          ;Params IlfProvider=kukaroboter.basistech.inlineforms.movement.spline; Kuka.IsGlobalPoint=False; Kuka.PointName=P254; Kuka.BlendingEnabled=False; Kuka.MoveDataName=CPDAT32; Kuka.VelocityPath=0.1; Kuka.VelocityFieldEnabled=True; Kuka.ColDetectFieldEnabled=True; Kuka.CurrentCDSetIndex=0; Kuka.MovementParameterFieldEnabled=True; IlfCommand=SLIN
          ;ENDFOLD
          SLIN XP254 WITH $VEL = SVEL_CP(0.1, , LCPDAT32), $TOOL = STOOL2(FP254), $BASE = SBASE(FP254.BASE_NO), $IPO_MODE = SIPO_MODE(FP254.IPO_FRAME), $LOAD = SLOAD(FP254.TOOL_NO), $ACC = SACC_CP(LCPDAT32), $ORI_TYPE = SORI_TYP(LCPDAT32), $APO = SAPO(LCPDAT32), $JERK = SJERK(LCPDAT32), $COLLMON_TOL_PRO[1] = USE_CM_PRO_VALUES(0)
          ;ENDFOLD
          ;FOLD Gripper SET [1]Gripper1 State=[2]CERRADA Wait 0.2[s] Check with Strategy 1 ;%{PE}
          ;FOLD Parameters Parameters ;%{h}
          ;Params IlfProvider=GripperTech.GripperSet;setgripper=1;setstate=2;setcont=nocont;waittime=0.2;errorstrategy=1
          ;ENDFOLD
          GRPg_SetStateAndCheck(1, 2, 0.2, 1)
          ;ENDFOLDinitialPosition
          ;FOLD SLIN P154 Vel=0.1 m/s CPDAT33 Tool[1]:SMC Base[0] ;%{PE}
          ;FOLD Parameters ;%{h}s
          ;Params IlfProvider=kukaroboter.basistech.inlineforms.movement.spline; Kuka.IsGlobalPoint=False; Kuka.PointName=P154; Kuka.BlendingEnabled=False; Kuka.MoveDataName=CPDAT33; Kuka.VelocityPath=0.1; Kuka.VelocityFieldEnabled=True; Kuka.ColDetectFieldEnabled=True; Kuka.CurrentCDSetIndex=0; Kuka.MovementParameterFieldEnabled=True; IlfCommand=SLIN
          ;ENDFOLD
          SLIN XP154 WITH $VEL = SVEL_CP(0.1, , LCPDAT33), $TOOL = STOOL2(FP154), $BASE = SBASE(FP154.BASE_NO), $IPO_MODE = SIPO_MODE(FP154.IPO_FRAME), $LOAD = SLOAD(FP154.TOOL_NO), $ACC = SACC_CP(LCPDAT33), $ORI_TYPE = SORI_TYP(LCPDAT33), $APO = SAPO(LCPDAT33), $JERK = SJERK(LCPDAT33), $COLLMON_TOL_PRO[1] = USE_CM_PRO_VALUES(0)
          ;ENDFOLD
          ;FOLD SPTP P500 Vel=100 % PDAT19 Tool[1]:SMC Base[0] ;%{PE}
          ;FOLD Parameters ;%{h}
          ;Params IlfProvider=kukaroboter.basistech.inlineforms.movement.spline; Kuka.IsGlobalPoint=False; Kuka.PointName=P500; Kuka.BlendingEnabled=False; Kuka.MoveDataPtpName=PDAT19; Kuka.VelocityPtp=100; Kuka.VelocityFieldEnabled=True; Kuka.ColDetectFieldEnabled=True; Kuka.CurrentCDSetIndex=0; Kuka.MovementParameterFieldEnabled=True; IlfCommand=SPTP
          ;ENDFOLD
          SPTP XP500 WITH $VEL_AXIS[1] = SVEL_JOINT(100.0), $TOOL = STOOL2(FP500), $BASE = SBASE(FP500.BASE_NO), $IPO_MODE = SIPO_MODE(FP500.IPO_FRAME), $LOAD = SLOAD(FP500.TOOL_NO), $ACC_AXIS[1] = SACC_JOINT(PPDAT19), $APO = SAPO_PTP(PPDAT19), $GEAR_JERK[1] = SGEAR_JERK(PPDAT19), $COLLMON_TOL_PRO[1] = USE_CM_PRO_VALUES(0)
          ;ENDFOLD
          ;FOLD Gripper SET [1]Gripper1 State=[1]ABIERTA Wait 0.2[s] Check with Strategy 1 ;%{PE}
          ;FOLD Parameters Parameters ;%{h}
          ;Params IlfProvider=GripperTech.GripperSet;setgripper=1;setstate=1;setcont=nocont;waittime=0.2;errorstrategy=1
          ;ENDFOLD
          GRPg_SetStateAndCheck(1, 1, 0.2, 1)
          ;ENDFOLD
      ENDIF
      IF eatPosition == 55 THEN
          ;FOLD SPTP P155 Vel=100 % PDAT1 Tool[1]:SMC Base[0] ;%{PE}
          ;FOLD Parameters ;%{h}
          ;Params IlfProvider=kukaroboter.basistech.inlineforms.movement.spline; Kuka.IsGlobalPoint=False; Kuka.PointName=P155; Kuka.BlendingEnabled=False; Kuka.MoveDataPtpName=PDAT1; Kuka.VelocityPtp=100; Kuka.VelocityFieldEnabled=True; Kuka.ColDetectFieldEnabled=True; Kuka.CurrentCDSetIndex=0; Kuka.MovementParameterFieldEnabled=True; IlfCommand=SPTP
          ;ENDFOLD
          SPTP XP155 WITH $VEL_AXIS[1] = SVEL_JOINT(100.0), $TOOL = STOOL2(FP155), $BASE = SBASE(FP155.BASE_NO), $IPO_MODE = SIPO_MODE(FP155.IPO_FRAME), $LOAD = SLOAD(FP155.TOOL_NO), $ACC_AXIS[1] = SACC_JOINT(PPDAT1), $APO = SAPO_PTP(PPDAT1), $GEAR_JERK[1] = SGEAR_JERK(PPDAT1), $COLLMON_TOL_PRO[1] = USE_CM_PRO_VALUES(0)
          ;ENDFOLD
          ;FOLD SLIN P255 Vel=0.1 m/s CPDAT32 Tool[1]:SMC Base[0] ;%{PE}
          ;FOLD Parameters ;%{h}
          ;Params IlfProvider=kukaroboter.basistech.inlineforms.movement.spline; Kuka.IsGlobalPoint=False; Kuka.PointName=P255; Kuka.BlendingEnabled=False; Kuka.MoveDataName=CPDAT32; Kuka.VelocityPath=0.1; Kuka.VelocityFieldEnabled=True; Kuka.ColDetectFieldEnabled=True; Kuka.CurrentCDSetIndex=0; Kuka.MovementParameterFieldEnabled=True; IlfCommand=SLIN
          ;ENDFOLD
          SLIN XP255 WITH $VEL = SVEL_CP(0.1, , LCPDAT32), $TOOL = STOOL2(FP255), $BASE = SBASE(FP255.BASE_NO), $IPO_MODE = SIPO_MODE(FP255.IPO_FRAME), $LOAD = SLOAD(FP255.TOOL_NO), $ACC = SACC_CP(LCPDAT32), $ORI_TYPE = SORI_TYP(LCPDAT32), $APO = SAPO(LCPDAT32), $JERK = SJERK(LCPDAT32), $COLLMON_TOL_PRO[1] = USE_CM_PRO_VALUES(0)
          ;ENDFOLD
          ;FOLD Gripper SET [1]Gripper1 State=[2]CERRADA Wait 0.2[s] Check with Strategy 1 ;%{PE}
          ;FOLD Parameters Parameters ;%{h}
          ;Params IlfProvider=GripperTech.GripperSet;setgripper=1;setstate=2;setcont=nocont;waittime=0.2;errorstrategy=1
          ;ENDFOLD
          GRPg_SetStateAndCheck(1, 2, 0.2, 1)
          ;ENDFOLDinitialPosition
          ;FOLD SLIN P155 Vel=0.1 m/s CPDAT33 Tool[1]:SMC Base[0] ;%{PE}
          ;FOLD Parameters ;%{h}s
          ;Params IlfProvider=kukaroboter.basistech.inlineforms.movement.spline; Kuka.IsGlobalPoint=False; Kuka.PointName=P155; Kuka.BlendingEnabled=False; Kuka.MoveDataName=CPDAT33; Kuka.VelocityPath=0.1; Kuka.VelocityFieldEnabled=True; Kuka.ColDetectFieldEnabled=True; Kuka.CurrentCDSetIndex=0; Kuka.MovementParameterFieldEnabled=True; IlfCommand=SLIN
          ;ENDFOLD
          SLIN XP155 WITH $VEL = SVEL_CP(0.1, , LCPDAT33), $TOOL = STOOL2(FP155), $BASE = SBASE(FP155.BASE_NO), $IPO_MODE = SIPO_MODE(FP155.IPO_FRAME), $LOAD = SLOAD(FP155.TOOL_NO), $ACC = SACC_CP(LCPDAT33), $ORI_TYPE = SORI_TYP(LCPDAT33), $APO = SAPO(LCPDAT33), $JERK = SJERK(LCPDAT33), $COLLMON_TOL_PRO[1] = USE_CM_PRO_VALUES(0)
          ;ENDFOLD
          ;FOLD SPTP P500 Vel=100 % PDAT19 Tool[1]:SMC Base[0] ;%{PE}
          ;FOLD Parameters ;%{h}
          ;Params IlfProvider=kukaroboter.basistech.inlineforms.movement.spline; Kuka.IsGlobalPoint=False; Kuka.PointName=P500; Kuka.BlendingEnabled=False; Kuka.MoveDataPtpName=PDAT19; Kuka.VelocityPtp=100; Kuka.VelocityFieldEnabled=True; Kuka.ColDetectFieldEnabled=True; Kuka.CurrentCDSetIndex=0; Kuka.MovementParameterFieldEnabled=True; IlfCommand=SPTP
          ;ENDFOLD
          SPTP XP500 WITH $VEL_AXIS[1] = SVEL_JOINT(100.0), $TOOL = STOOL2(FP500), $BASE = SBASE(FP500.BASE_NO), $IPO_MODE = SIPO_MODE(FP500.IPO_FRAME), $LOAD = SLOAD(FP500.TOOL_NO), $ACC_AXIS[1] = SACC_JOINT(PPDAT19), $APO = SAPO_PTP(PPDAT19), $GEAR_JERK[1] = SGEAR_JERK(PPDAT19), $COLLMON_TOL_PRO[1] = USE_CM_PRO_VALUES(0)
          ;ENDFOLD
          ;FOLD Gripper SET [1]Gripper1 State=[1]ABIERTA Wait 0.2[s] Check with Strategy 1 ;%{PE}
          ;FOLD Parameters Parameters ;%{h}
          ;Params IlfProvider=GripperTech.GripperSet;setgripper=1;setstate=1;setcont=nocont;waittime=0.2;errorstrategy=1
          ;ENDFOLD
          GRPg_SetStateAndCheck(1, 1, 0.2, 1)
          ;ENDFOLD
      ENDIF
      IF eatPosition == 56 THEN
          ;FOLD SPTP P156 Vel=100 % PDAT1 Tool[1]:SMC Base[0] ;%{PE}
          ;FOLD Parameters ;%{h}
          ;Params IlfProvider=kukaroboter.basistech.inlineforms.movement.spline; Kuka.IsGlobalPoint=False; Kuka.PointName=P156; Kuka.BlendingEnabled=False; Kuka.MoveDataPtpName=PDAT1; Kuka.VelocityPtp=100; Kuka.VelocityFieldEnabled=True; Kuka.ColDetectFieldEnabled=True; Kuka.CurrentCDSetIndex=0; Kuka.MovementParameterFieldEnabled=True; IlfCommand=SPTP
          ;ENDFOLD
          SPTP XP156 WITH $VEL_AXIS[1] = SVEL_JOINT(100.0), $TOOL = STOOL2(FP156), $BASE = SBASE(FP156.BASE_NO), $IPO_MODE = SIPO_MODE(FP156.IPO_FRAME), $LOAD = SLOAD(FP156.TOOL_NO), $ACC_AXIS[1] = SACC_JOINT(PPDAT1), $APO = SAPO_PTP(PPDAT1), $GEAR_JERK[1] = SGEAR_JERK(PPDAT1), $COLLMON_TOL_PRO[1] = USE_CM_PRO_VALUES(0)
          ;ENDFOLD
          ;FOLD SLIN P256 Vel=0.1 m/s CPDAT32 Tool[1]:SMC Base[0] ;%{PE}
          ;FOLD Parameters ;%{h}
          ;Params IlfProvider=kukaroboter.basistech.inlineforms.movement.spline; Kuka.IsGlobalPoint=False; Kuka.PointName=P256; Kuka.BlendingEnabled=False; Kuka.MoveDataName=CPDAT32; Kuka.VelocityPath=0.1; Kuka.VelocityFieldEnabled=True; Kuka.ColDetectFieldEnabled=True; Kuka.CurrentCDSetIndex=0; Kuka.MovementParameterFieldEnabled=True; IlfCommand=SLIN
          ;ENDFOLD
          SLIN XP256 WITH $VEL = SVEL_CP(0.1, , LCPDAT32), $TOOL = STOOL2(FP256), $BASE = SBASE(FP256.BASE_NO), $IPO_MODE = SIPO_MODE(FP256.IPO_FRAME), $LOAD = SLOAD(FP256.TOOL_NO), $ACC = SACC_CP(LCPDAT32), $ORI_TYPE = SORI_TYP(LCPDAT32), $APO = SAPO(LCPDAT32), $JERK = SJERK(LCPDAT32), $COLLMON_TOL_PRO[1] = USE_CM_PRO_VALUES(0)
          ;ENDFOLD
          ;FOLD Gripper SET [1]Gripper1 State=[2]CERRADA Wait 0.2[s] Check with Strategy 1 ;%{PE}
          ;FOLD Parameters Parameters ;%{h}
          ;Params IlfProvider=GripperTech.GripperSet;setgripper=1;setstate=2;setcont=nocont;waittime=0.2;errorstrategy=1
          ;ENDFOLD
          GRPg_SetStateAndCheck(1, 2, 0.2, 1)
          ;ENDFOLDinitialPosition
          ;FOLD SLIN P156 Vel=0.1 m/s CPDAT33 Tool[1]:SMC Base[0] ;%{PE}
          ;FOLD Parameters ;%{h}s
          ;Params IlfProvider=kukaroboter.basistech.inlineforms.movement.spline; Kuka.IsGlobalPoint=False; Kuka.PointName=P156; Kuka.BlendingEnabled=False; Kuka.MoveDataName=CPDAT33; Kuka.VelocityPath=0.1; Kuka.VelocityFieldEnabled=True; Kuka.ColDetectFieldEnabled=True; Kuka.CurrentCDSetIndex=0; Kuka.MovementParameterFieldEnabled=True; IlfCommand=SLIN
          ;ENDFOLD
          SLIN XP156 WITH $VEL = SVEL_CP(0.1, , LCPDAT33), $TOOL = STOOL2(FP156), $BASE = SBASE(FP156.BASE_NO), $IPO_MODE = SIPO_MODE(FP156.IPO_FRAME), $LOAD = SLOAD(FP156.TOOL_NO), $ACC = SACC_CP(LCPDAT33), $ORI_TYPE = SORI_TYP(LCPDAT33), $APO = SAPO(LCPDAT33), $JERK = SJERK(LCPDAT33), $COLLMON_TOL_PRO[1] = USE_CM_PRO_VALUES(0)
          ;ENDFOLD
          ;FOLD SPTP P500 Vel=100 % PDAT19 Tool[1]:SMC Base[0] ;%{PE}
          ;FOLD Parameters ;%{h}
          ;Params IlfProvider=kukaroboter.basistech.inlineforms.movement.spline; Kuka.IsGlobalPoint=False; Kuka.PointName=P500; Kuka.BlendingEnabled=False; Kuka.MoveDataPtpName=PDAT19; Kuka.VelocityPtp=100; Kuka.VelocityFieldEnabled=True; Kuka.ColDetectFieldEnabled=True; Kuka.CurrentCDSetIndex=0; Kuka.MovementParameterFieldEnabled=True; IlfCommand=SPTP
          ;ENDFOLD
          SPTP XP500 WITH $VEL_AXIS[1] = SVEL_JOINT(100.0), $TOOL = STOOL2(FP500), $BASE = SBASE(FP500.BASE_NO), $IPO_MODE = SIPO_MODE(FP500.IPO_FRAME), $LOAD = SLOAD(FP500.TOOL_NO), $ACC_AXIS[1] = SACC_JOINT(PPDAT19), $APO = SAPO_PTP(PPDAT19), $GEAR_JERK[1] = SGEAR_JERK(PPDAT19), $COLLMON_TOL_PRO[1] = USE_CM_PRO_VALUES(0)
          ;ENDFOLD
          ;FOLD Gripper SET [1]Gripper1 State=[1]ABIERTA Wait 0.2[s] Check with Strategy 1 ;%{PE}
          ;FOLD Parameters Parameters ;%{h}
          ;Params IlfProvider=GripperTech.GripperSet;setgripper=1;setstate=1;setcont=nocont;waittime=0.2;errorstrategy=1
          ;ENDFOLD
          GRPg_SetStateAndCheck(1, 1, 0.2, 1)
          ;ENDFOLD
      ENDIF
      IF eatPosition == 57 THEN
          ;FOLD SPTP P157 Vel=100 % PDAT1 Tool[1]:SMC Base[0] ;%{PE}
          ;FOLD Parameters ;%{h}
          ;Params IlfProvider=kukaroboter.basistech.inlineforms.movement.spline; Kuka.IsGlobalPoint=False; Kuka.PointName=P157; Kuka.BlendingEnabled=False; Kuka.MoveDataPtpName=PDAT1; Kuka.VelocityPtp=100; Kuka.VelocityFieldEnabled=True; Kuka.ColDetectFieldEnabled=True; Kuka.CurrentCDSetIndex=0; Kuka.MovementParameterFieldEnabled=True; IlfCommand=SPTP
          ;ENDFOLD
          SPTP XP157 WITH $VEL_AXIS[1] = SVEL_JOINT(100.0), $TOOL = STOOL2(FP157), $BASE = SBASE(FP157.BASE_NO), $IPO_MODE = SIPO_MODE(FP157.IPO_FRAME), $LOAD = SLOAD(FP157.TOOL_NO), $ACC_AXIS[1] = SACC_JOINT(PPDAT1), $APO = SAPO_PTP(PPDAT1), $GEAR_JERK[1] = SGEAR_JERK(PPDAT1), $COLLMON_TOL_PRO[1] = USE_CM_PRO_VALUES(0)
          ;ENDFOLD
          ;FOLD SLIN P257 Vel=0.1 m/s CPDAT32 Tool[1]:SMC Base[0] ;%{PE}
          ;FOLD Parameters ;%{h}
          ;Params IlfProvider=kukaroboter.basistech.inlineforms.movement.spline; Kuka.IsGlobalPoint=False; Kuka.PointName=P257; Kuka.BlendingEnabled=False; Kuka.MoveDataName=CPDAT32; Kuka.VelocityPath=0.1; Kuka.VelocityFieldEnabled=True; Kuka.ColDetectFieldEnabled=True; Kuka.CurrentCDSetIndex=0; Kuka.MovementParameterFieldEnabled=True; IlfCommand=SLIN
          ;ENDFOLD
          SLIN XP257 WITH $VEL = SVEL_CP(0.1, , LCPDAT32), $TOOL = STOOL2(FP257), $BASE = SBASE(FP257.BASE_NO), $IPO_MODE = SIPO_MODE(FP257.IPO_FRAME), $LOAD = SLOAD(FP257.TOOL_NO), $ACC = SACC_CP(LCPDAT32), $ORI_TYPE = SORI_TYP(LCPDAT32), $APO = SAPO(LCPDAT32), $JERK = SJERK(LCPDAT32), $COLLMON_TOL_PRO[1] = USE_CM_PRO_VALUES(0)
          ;ENDFOLD
          ;FOLD Gripper SET [1]Gripper1 State=[2]CERRADA Wait 0.2[s] Check with Strategy 1 ;%{PE}
          ;FOLD Parameters Parameters ;%{h}
          ;Params IlfProvider=GripperTech.GripperSet;setgripper=1;setstate=2;setcont=nocont;waittime=0.2;errorstrategy=1
          ;ENDFOLD
          GRPg_SetStateAndCheck(1, 2, 0.2, 1)
          ;ENDFOLDinitialPosition
          ;FOLD SLIN P157 Vel=0.1 m/s CPDAT33 Tool[1]:SMC Base[0] ;%{PE}
          ;FOLD Parameters ;%{h}s
          ;Params IlfProvider=kukaroboter.basistech.inlineforms.movement.spline; Kuka.IsGlobalPoint=False; Kuka.PointName=P157; Kuka.BlendingEnabled=False; Kuka.MoveDataName=CPDAT33; Kuka.VelocityPath=0.1; Kuka.VelocityFieldEnabled=True; Kuka.ColDetectFieldEnabled=True; Kuka.CurrentCDSetIndex=0; Kuka.MovementParameterFieldEnabled=True; IlfCommand=SLIN
          ;ENDFOLD
          SLIN XP157 WITH $VEL = SVEL_CP(0.1, , LCPDAT33), $TOOL = STOOL2(FP157), $BASE = SBASE(FP157.BASE_NO), $IPO_MODE = SIPO_MODE(FP157.IPO_FRAME), $LOAD = SLOAD(FP157.TOOL_NO), $ACC = SACC_CP(LCPDAT33), $ORI_TYPE = SORI_TYP(LCPDAT33), $APO = SAPO(LCPDAT33), $JERK = SJERK(LCPDAT33), $COLLMON_TOL_PRO[1] = USE_CM_PRO_VALUES(0)
          ;ENDFOLD
          ;FOLD SPTP P500 Vel=100 % PDAT19 Tool[1]:SMC Base[0] ;%{PE}
          ;FOLD Parameters ;%{h}
          ;Params IlfProvider=kukaroboter.basistech.inlineforms.movement.spline; Kuka.IsGlobalPoint=False; Kuka.PointName=P500; Kuka.BlendingEnabled=False; Kuka.MoveDataPtpName=PDAT19; Kuka.VelocityPtp=100; Kuka.VelocityFieldEnabled=True; Kuka.ColDetectFieldEnabled=True; Kuka.CurrentCDSetIndex=0; Kuka.MovementParameterFieldEnabled=True; IlfCommand=SPTP
          ;ENDFOLD
          SPTP XP500 WITH $VEL_AXIS[1] = SVEL_JOINT(100.0), $TOOL = STOOL2(FP500), $BASE = SBASE(FP500.BASE_NO), $IPO_MODE = SIPO_MODE(FP500.IPO_FRAME), $LOAD = SLOAD(FP500.TOOL_NO), $ACC_AXIS[1] = SACC_JOINT(PPDAT19), $APO = SAPO_PTP(PPDAT19), $GEAR_JERK[1] = SGEAR_JERK(PPDAT19), $COLLMON_TOL_PRO[1] = USE_CM_PRO_VALUES(0)
          ;ENDFOLD
          ;FOLD Gripper SET [1]Gripper1 State=[1]ABIERTA Wait 0.2[s] Check with Strategy 1 ;%{PE}
          ;FOLD Parameters Parameters ;%{h}
          ;Params IlfProvider=GripperTech.GripperSet;setgripper=1;setstate=1;setcont=nocont;waittime=0.2;errorstrategy=1
          ;ENDFOLD
          GRPg_SetStateAndCheck(1, 1, 0.2, 1)
          ;ENDFOLD
      ENDIF
      IF eatPosition == 58 THEN
          ;FOLD SPTP P158 Vel=100 % PDAT1 Tool[1]:SMC Base[0] ;%{PE}
          ;FOLD Parameters ;%{h}
          ;Params IlfProvider=kukaroboter.basistech.inlineforms.movement.spline; Kuka.IsGlobalPoint=False; Kuka.PointName=P158; Kuka.BlendingEnabled=False; Kuka.MoveDataPtpName=PDAT1; Kuka.VelocityPtp=100; Kuka.VelocityFieldEnabled=True; Kuka.ColDetectFieldEnabled=True; Kuka.CurrentCDSetIndex=0; Kuka.MovementParameterFieldEnabled=True; IlfCommand=SPTP
          ;ENDFOLD
          SPTP XP158 WITH $VEL_AXIS[1] = SVEL_JOINT(100.0), $TOOL = STOOL2(FP158), $BASE = SBASE(FP158.BASE_NO), $IPO_MODE = SIPO_MODE(FP158.IPO_FRAME), $LOAD = SLOAD(FP158.TOOL_NO), $ACC_AXIS[1] = SACC_JOINT(PPDAT1), $APO = SAPO_PTP(PPDAT1), $GEAR_JERK[1] = SGEAR_JERK(PPDAT1), $COLLMON_TOL_PRO[1] = USE_CM_PRO_VALUES(0)
          ;ENDFOLD
          ;FOLD SLIN P258 Vel=0.1 m/s CPDAT32 Tool[1]:SMC Base[0] ;%{PE}
          ;FOLD Parameters ;%{h}
          ;Params IlfProvider=kukaroboter.basistech.inlineforms.movement.spline; Kuka.IsGlobalPoint=False; Kuka.PointName=P258; Kuka.BlendingEnabled=False; Kuka.MoveDataName=CPDAT32; Kuka.VelocityPath=0.1; Kuka.VelocityFieldEnabled=True; Kuka.ColDetectFieldEnabled=True; Kuka.CurrentCDSetIndex=0; Kuka.MovementParameterFieldEnabled=True; IlfCommand=SLIN
          ;ENDFOLD
          SLIN XP258 WITH $VEL = SVEL_CP(0.1, , LCPDAT32), $TOOL = STOOL2(FP258), $BASE = SBASE(FP258.BASE_NO), $IPO_MODE = SIPO_MODE(FP258.IPO_FRAME), $LOAD = SLOAD(FP258.TOOL_NO), $ACC = SACC_CP(LCPDAT32), $ORI_TYPE = SORI_TYP(LCPDAT32), $APO = SAPO(LCPDAT32), $JERK = SJERK(LCPDAT32), $COLLMON_TOL_PRO[1] = USE_CM_PRO_VALUES(0)
          ;ENDFOLD
          ;FOLD Gripper SET [1]Gripper1 State=[2]CERRADA Wait 0.2[s] Check with Strategy 1 ;%{PE}
          ;FOLD Parameters Parameters ;%{h}
          ;Params IlfProvider=GripperTech.GripperSet;setgripper=1;setstate=2;setcont=nocont;waittime=0.2;errorstrategy=1
          ;ENDFOLD
          GRPg_SetStateAndCheck(1, 2, 0.2, 1)
          ;ENDFOLDinitialPosition
          ;FOLD SLIN P158 Vel=0.1 m/s CPDAT33 Tool[1]:SMC Base[0] ;%{PE}
          ;FOLD Parameters ;%{h}s
          ;Params IlfProvider=kukaroboter.basistech.inlineforms.movement.spline; Kuka.IsGlobalPoint=False; Kuka.PointName=P158; Kuka.BlendingEnabled=False; Kuka.MoveDataName=CPDAT33; Kuka.VelocityPath=0.1; Kuka.VelocityFieldEnabled=True; Kuka.ColDetectFieldEnabled=True; Kuka.CurrentCDSetIndex=0; Kuka.MovementParameterFieldEnabled=True; IlfCommand=SLIN
          ;ENDFOLD
          SLIN XP158 WITH $VEL = SVEL_CP(0.1, , LCPDAT33), $TOOL = STOOL2(FP158), $BASE = SBASE(FP158.BASE_NO), $IPO_MODE = SIPO_MODE(FP158.IPO_FRAME), $LOAD = SLOAD(FP158.TOOL_NO), $ACC = SACC_CP(LCPDAT33), $ORI_TYPE = SORI_TYP(LCPDAT33), $APO = SAPO(LCPDAT33), $JERK = SJERK(LCPDAT33), $COLLMON_TOL_PRO[1] = USE_CM_PRO_VALUES(0)
          ;ENDFOLD
          ;FOLD SPTP P500 Vel=100 % PDAT19 Tool[1]:SMC Base[0] ;%{PE}
          ;FOLD Parameters ;%{h}
          ;Params IlfProvider=kukaroboter.basistech.inlineforms.movement.spline; Kuka.IsGlobalPoint=False; Kuka.PointName=P500; Kuka.BlendingEnabled=False; Kuka.MoveDataPtpName=PDAT19; Kuka.VelocityPtp=100; Kuka.VelocityFieldEnabled=True; Kuka.ColDetectFieldEnabled=True; Kuka.CurrentCDSetIndex=0; Kuka.MovementParameterFieldEnabled=True; IlfCommand=SPTP
          ;ENDFOLD
          SPTP XP500 WITH $VEL_AXIS[1] = SVEL_JOINT(100.0), $TOOL = STOOL2(FP500), $BASE = SBASE(FP500.BASE_NO), $IPO_MODE = SIPO_MODE(FP500.IPO_FRAME), $LOAD = SLOAD(FP500.TOOL_NO), $ACC_AXIS[1] = SACC_JOINT(PPDAT19), $APO = SAPO_PTP(PPDAT19), $GEAR_JERK[1] = SGEAR_JERK(PPDAT19), $COLLMON_TOL_PRO[1] = USE_CM_PRO_VALUES(0)
          ;ENDFOLD
          ;FOLD Gripper SET [1]Gripper1 State=[1]ABIERTA Wait 0.2[s] Check with Strategy 1 ;%{PE}
          ;FOLD Parameters Parameters ;%{h}
          ;Params IlfProvider=GripperTech.GripperSet;setgripper=1;setstate=1;setcont=nocont;waittime=0.2;errorstrategy=1
          ;ENDFOLD
          GRPg_SetStateAndCheck(1, 1, 0.2, 1)
          ;ENDFOLD
      ENDIF
      IF eatPosition == 59 THEN
          ;FOLD SPTP P159 Vel=100 % PDAT1 Tool[1]:SMC Base[0] ;%{PE}
          ;FOLD Parameters ;%{h}
          ;Params IlfProvider=kukaroboter.basistech.inlineforms.movement.spline; Kuka.IsGlobalPoint=False; Kuka.PointName=P159; Kuka.BlendingEnabled=False; Kuka.MoveDataPtpName=PDAT1; Kuka.VelocityPtp=100; Kuka.VelocityFieldEnabled=True; Kuka.ColDetectFieldEnabled=True; Kuka.CurrentCDSetIndex=0; Kuka.MovementParameterFieldEnabled=True; IlfCommand=SPTP
          ;ENDFOLD
          SPTP XP159 WITH $VEL_AXIS[1] = SVEL_JOINT(100.0), $TOOL = STOOL2(FP159), $BASE = SBASE(FP159.BASE_NO), $IPO_MODE = SIPO_MODE(FP159.IPO_FRAME), $LOAD = SLOAD(FP159.TOOL_NO), $ACC_AXIS[1] = SACC_JOINT(PPDAT1), $APO = SAPO_PTP(PPDAT1), $GEAR_JERK[1] = SGEAR_JERK(PPDAT1), $COLLMON_TOL_PRO[1] = USE_CM_PRO_VALUES(0)
          ;ENDFOLD
          ;FOLD SLIN P259 Vel=0.1 m/s CPDAT32 Tool[1]:SMC Base[0] ;%{PE}
          ;FOLD Parameters ;%{h}
          ;Params IlfProvider=kukaroboter.basistech.inlineforms.movement.spline; Kuka.IsGlobalPoint=False; Kuka.PointName=P259; Kuka.BlendingEnabled=False; Kuka.MoveDataName=CPDAT32; Kuka.VelocityPath=0.1; Kuka.VelocityFieldEnabled=True; Kuka.ColDetectFieldEnabled=True; Kuka.CurrentCDSetIndex=0; Kuka.MovementParameterFieldEnabled=True; IlfCommand=SLIN
          ;ENDFOLD
          SLIN XP259 WITH $VEL = SVEL_CP(0.1, , LCPDAT32), $TOOL = STOOL2(FP259), $BASE = SBASE(FP259.BASE_NO), $IPO_MODE = SIPO_MODE(FP259.IPO_FRAME), $LOAD = SLOAD(FP259.TOOL_NO), $ACC = SACC_CP(LCPDAT32), $ORI_TYPE = SORI_TYP(LCPDAT32), $APO = SAPO(LCPDAT32), $JERK = SJERK(LCPDAT32), $COLLMON_TOL_PRO[1] = USE_CM_PRO_VALUES(0)
          ;ENDFOLD
          ;FOLD Gripper SET [1]Gripper1 State=[2]CERRADA Wait 0.2[s] Check with Strategy 1 ;%{PE}
          ;FOLD Parameters Parameters ;%{h}
          ;Params IlfProvider=GripperTech.GripperSet;setgripper=1;setstate=2;setcont=nocont;waittime=0.2;errorstrategy=1
          ;ENDFOLD
          GRPg_SetStateAndCheck(1, 2, 0.2, 1)
          ;ENDFOLDinitialPosition
          ;FOLD SLIN P159 Vel=0.1 m/s CPDAT33 Tool[1]:SMC Base[0] ;%{PE}
          ;FOLD Parameters ;%{h}s
          ;Params IlfProvider=kukaroboter.basistech.inlineforms.movement.spline; Kuka.IsGlobalPoint=False; Kuka.PointName=P159; Kuka.BlendingEnabled=False; Kuka.MoveDataName=CPDAT33; Kuka.VelocityPath=0.1; Kuka.VelocityFieldEnabled=True; Kuka.ColDetectFieldEnabled=True; Kuka.CurrentCDSetIndex=0; Kuka.MovementParameterFieldEnabled=True; IlfCommand=SLIN
          ;ENDFOLD
          SLIN XP159 WITH $VEL = SVEL_CP(0.1, , LCPDAT33), $TOOL = STOOL2(FP159), $BASE = SBASE(FP159.BASE_NO), $IPO_MODE = SIPO_MODE(FP159.IPO_FRAME), $LOAD = SLOAD(FP159.TOOL_NO), $ACC = SACC_CP(LCPDAT33), $ORI_TYPE = SORI_TYP(LCPDAT33), $APO = SAPO(LCPDAT33), $JERK = SJERK(LCPDAT33), $COLLMON_TOL_PRO[1] = USE_CM_PRO_VALUES(0)
          ;ENDFOLD
          ;FOLD SPTP P500 Vel=100 % PDAT19 Tool[1]:SMC Base[0] ;%{PE}
          ;FOLD Parameters ;%{h}
          ;Params IlfProvider=kukaroboter.basistech.inlineforms.movement.spline; Kuka.IsGlobalPoint=False; Kuka.PointName=P500; Kuka.BlendingEnabled=False; Kuka.MoveDataPtpName=PDAT19; Kuka.VelocityPtp=100; Kuka.VelocityFieldEnabled=True; Kuka.ColDetectFieldEnabled=True; Kuka.CurrentCDSetIndex=0; Kuka.MovementParameterFieldEnabled=True; IlfCommand=SPTP
          ;ENDFOLD
          SPTP XP500 WITH $VEL_AXIS[1] = SVEL_JOINT(100.0), $TOOL = STOOL2(FP500), $BASE = SBASE(FP500.BASE_NO), $IPO_MODE = SIPO_MODE(FP500.IPO_FRAME), $LOAD = SLOAD(FP500.TOOL_NO), $ACC_AXIS[1] = SACC_JOINT(PPDAT19), $APO = SAPO_PTP(PPDAT19), $GEAR_JERK[1] = SGEAR_JERK(PPDAT19), $COLLMON_TOL_PRO[1] = USE_CM_PRO_VALUES(0)
          ;ENDFOLD
          ;FOLD Gripper SET [1]Gripper1 State=[1]ABIERTA Wait 0.2[s] Check with Strategy 1 ;%{PE}
          ;FOLD Parameters Parameters ;%{h}
          ;Params IlfProvider=GripperTech.GripperSet;setgripper=1;setstate=1;setcont=nocont;waittime=0.2;errorstrategy=1
          ;ENDFOLD
          GRPg_SetStateAndCheck(1, 1, 0.2, 1)
          ;ENDFOLD
      ENDIF
      IF eatPosition == 60 THEN
          ;FOLD SPTP P160 Vel=100 % PDAT1 Tool[1]:SMC Base[0] ;%{PE}
          ;FOLD Parameters ;%{h}
          ;Params IlfProvider=kukaroboter.basistech.inlineforms.movement.spline; Kuka.IsGlobalPoint=False; Kuka.PointName=P160; Kuka.BlendingEnabled=False; Kuka.MoveDataPtpName=PDAT1; Kuka.VelocityPtp=100; Kuka.VelocityFieldEnabled=True; Kuka.ColDetectFieldEnabled=True; Kuka.CurrentCDSetIndex=0; Kuka.MovementParameterFieldEnabled=True; IlfCommand=SPTP
          ;ENDFOLD
          SPTP XP160 WITH $VEL_AXIS[1] = SVEL_JOINT(100.0), $TOOL = STOOL2(FP160), $BASE = SBASE(FP160.BASE_NO), $IPO_MODE = SIPO_MODE(FP160.IPO_FRAME), $LOAD = SLOAD(FP160.TOOL_NO), $ACC_AXIS[1] = SACC_JOINT(PPDAT1), $APO = SAPO_PTP(PPDAT1), $GEAR_JERK[1] = SGEAR_JERK(PPDAT1), $COLLMON_TOL_PRO[1] = USE_CM_PRO_VALUES(0)
          ;ENDFOLD
          ;FOLD SLIN P260 Vel=0.1 m/s CPDAT32 Tool[1]:SMC Base[0] ;%{PE}
          ;FOLD Parameters ;%{h}
          ;Params IlfProvider=kukaroboter.basistech.inlineforms.movement.spline; Kuka.IsGlobalPoint=False; Kuka.PointName=P260; Kuka.BlendingEnabled=False; Kuka.MoveDataName=CPDAT32; Kuka.VelocityPath=0.1; Kuka.VelocityFieldEnabled=True; Kuka.ColDetectFieldEnabled=True; Kuka.CurrentCDSetIndex=0; Kuka.MovementParameterFieldEnabled=True; IlfCommand=SLIN
          ;ENDFOLD
          SLIN XP260 WITH $VEL = SVEL_CP(0.1, , LCPDAT32), $TOOL = STOOL2(FP260), $BASE = SBASE(FP260.BASE_NO), $IPO_MODE = SIPO_MODE(FP260.IPO_FRAME), $LOAD = SLOAD(FP260.TOOL_NO), $ACC = SACC_CP(LCPDAT32), $ORI_TYPE = SORI_TYP(LCPDAT32), $APO = SAPO(LCPDAT32), $JERK = SJERK(LCPDAT32), $COLLMON_TOL_PRO[1] = USE_CM_PRO_VALUES(0)
          ;ENDFOLD
          ;FOLD Gripper SET [1]Gripper1 State=[2]CERRADA Wait 0.2[s] Check with Strategy 1 ;%{PE}
          ;FOLD Parameters Parameters ;%{h}
          ;Params IlfProvider=GripperTech.GripperSet;setgripper=1;setstate=2;setcont=nocont;waittime=0.2;errorstrategy=1
          ;ENDFOLD
          GRPg_SetStateAndCheck(1, 2, 0.2, 1)
          ;ENDFOLDinitialPosition
          ;FOLD SLIN P160 Vel=0.1 m/s CPDAT33 Tool[1]:SMC Base[0] ;%{PE}
          ;FOLD Parameters ;%{h}s
          ;Params IlfProvider=kukaroboter.basistech.inlineforms.movement.spline; Kuka.IsGlobalPoint=False; Kuka.PointName=P160; Kuka.BlendingEnabled=False; Kuka.MoveDataName=CPDAT33; Kuka.VelocityPath=0.1; Kuka.VelocityFieldEnabled=True; Kuka.ColDetectFieldEnabled=True; Kuka.CurrentCDSetIndex=0; Kuka.MovementParameterFieldEnabled=True; IlfCommand=SLIN
          ;ENDFOLD
          SLIN XP160 WITH $VEL = SVEL_CP(0.1, , LCPDAT33), $TOOL = STOOL2(FP160), $BASE = SBASE(FP160.BASE_NO), $IPO_MODE = SIPO_MODE(FP160.IPO_FRAME), $LOAD = SLOAD(FP160.TOOL_NO), $ACC = SACC_CP(LCPDAT33), $ORI_TYPE = SORI_TYP(LCPDAT33), $APO = SAPO(LCPDAT33), $JERK = SJERK(LCPDAT33), $COLLMON_TOL_PRO[1] = USE_CM_PRO_VALUES(0)
          ;ENDFOLD
          ;FOLD SPTP P500 Vel=100 % PDAT19 Tool[1]:SMC Base[0] ;%{PE}
          ;FOLD Parameters ;%{h}
          ;Params IlfProvider=kukaroboter.basistech.inlineforms.movement.spline; Kuka.IsGlobalPoint=False; Kuka.PointName=P500; Kuka.BlendingEnabled=False; Kuka.MoveDataPtpName=PDAT19; Kuka.VelocityPtp=100; Kuka.VelocityFieldEnabled=True; Kuka.ColDetectFieldEnabled=True; Kuka.CurrentCDSetIndex=0; Kuka.MovementParameterFieldEnabled=True; IlfCommand=SPTP
          ;ENDFOLD
          SPTP XP500 WITH $VEL_AXIS[1] = SVEL_JOINT(100.0), $TOOL = STOOL2(FP500), $BASE = SBASE(FP500.BASE_NO), $IPO_MODE = SIPO_MODE(FP500.IPO_FRAME), $LOAD = SLOAD(FP500.TOOL_NO), $ACC_AXIS[1] = SACC_JOINT(PPDAT19), $APO = SAPO_PTP(PPDAT19), $GEAR_JERK[1] = SGEAR_JERK(PPDAT19), $COLLMON_TOL_PRO[1] = USE_CM_PRO_VALUES(0)
          ;ENDFOLD
          ;FOLD Gripper SET [1]Gripper1 State=[1]ABIERTA Wait 0.2[s] Check with Strategy 1 ;%{PE}
          ;FOLD Parameters Parameters ;%{h}
          ;Params IlfProvider=GripperTech.GripperSet;setgripper=1;setstate=1;setcont=nocont;waittime=0.2;errorstrategy=1
          ;ENDFOLD
          GRPg_SetStateAndCheck(1, 1, 0.2, 1)
          ;ENDFOLD
      ENDIF
      IF eatPosition == 61 THEN
          ;FOLD SPTP P161 Vel=100 % PDAT1 Tool[1]:SMC Base[0] ;%{PE}
          ;FOLD Parameters ;%{h}
          ;Params IlfProvider=kukaroboter.basistech.inlineforms.movement.spline; Kuka.IsGlobalPoint=False; Kuka.PointName=P161; Kuka.BlendingEnabled=False; Kuka.MoveDataPtpName=PDAT1; Kuka.VelocityPtp=100; Kuka.VelocityFieldEnabled=True; Kuka.ColDetectFieldEnabled=True; Kuka.CurrentCDSetIndex=0; Kuka.MovementParameterFieldEnabled=True; IlfCommand=SPTP
          ;ENDFOLD
          SPTP XP161 WITH $VEL_AXIS[1] = SVEL_JOINT(100.0), $TOOL = STOOL2(FP161), $BASE = SBASE(FP161.BASE_NO), $IPO_MODE = SIPO_MODE(FP161.IPO_FRAME), $LOAD = SLOAD(FP161.TOOL_NO), $ACC_AXIS[1] = SACC_JOINT(PPDAT1), $APO = SAPO_PTP(PPDAT1), $GEAR_JERK[1] = SGEAR_JERK(PPDAT1), $COLLMON_TOL_PRO[1] = USE_CM_PRO_VALUES(0)
          ;ENDFOLD
          ;FOLD SLIN P261 Vel=0.1 m/s CPDAT32 Tool[1]:SMC Base[0] ;%{PE}
          ;FOLD Parameters ;%{h}
          ;Params IlfProvider=kukaroboter.basistech.inlineforms.movement.spline; Kuka.IsGlobalPoint=False; Kuka.PointName=P261; Kuka.BlendingEnabled=False; Kuka.MoveDataName=CPDAT32; Kuka.VelocityPath=0.1; Kuka.VelocityFieldEnabled=True; Kuka.ColDetectFieldEnabled=True; Kuka.CurrentCDSetIndex=0; Kuka.MovementParameterFieldEnabled=True; IlfCommand=SLIN
          ;ENDFOLD
          SLIN XP261 WITH $VEL = SVEL_CP(0.1, , LCPDAT32), $TOOL = STOOL2(FP261), $BASE = SBASE(FP261.BASE_NO), $IPO_MODE = SIPO_MODE(FP261.IPO_FRAME), $LOAD = SLOAD(FP261.TOOL_NO), $ACC = SACC_CP(LCPDAT32), $ORI_TYPE = SORI_TYP(LCPDAT32), $APO = SAPO(LCPDAT32), $JERK = SJERK(LCPDAT32), $COLLMON_TOL_PRO[1] = USE_CM_PRO_VALUES(0)
          ;ENDFOLD
          ;FOLD Gripper SET [1]Gripper1 State=[2]CERRADA Wait 0.2[s] Check with Strategy 1 ;%{PE}
          ;FOLD Parameters Parameters ;%{h}
          ;Params IlfProvider=GripperTech.GripperSet;setgripper=1;setstate=2;setcont=nocont;waittime=0.2;errorstrategy=1
          ;ENDFOLD
          GRPg_SetStateAndCheck(1, 2, 0.2, 1)
          ;ENDFOLDinitialPosition
          ;FOLD SLIN P161 Vel=0.1 m/s CPDAT33 Tool[1]:SMC Base[0] ;%{PE}
          ;FOLD Parameters ;%{h}s
          ;Params IlfProvider=kukaroboter.basistech.inlineforms.movement.spline; Kuka.IsGlobalPoint=False; Kuka.PointName=P161; Kuka.BlendingEnabled=False; Kuka.MoveDataName=CPDAT33; Kuka.VelocityPath=0.1; Kuka.VelocityFieldEnabled=True; Kuka.ColDetectFieldEnabled=True; Kuka.CurrentCDSetIndex=0; Kuka.MovementParameterFieldEnabled=True; IlfCommand=SLIN
          ;ENDFOLD
          SLIN XP161 WITH $VEL = SVEL_CP(0.1, , LCPDAT33), $TOOL = STOOL2(FP161), $BASE = SBASE(FP161.BASE_NO), $IPO_MODE = SIPO_MODE(FP161.IPO_FRAME), $LOAD = SLOAD(FP161.TOOL_NO), $ACC = SACC_CP(LCPDAT33), $ORI_TYPE = SORI_TYP(LCPDAT33), $APO = SAPO(LCPDAT33), $JERK = SJERK(LCPDAT33), $COLLMON_TOL_PRO[1] = USE_CM_PRO_VALUES(0)
          ;ENDFOLD
          ;FOLD SPTP P500 Vel=100 % PDAT19 Tool[1]:SMC Base[0] ;%{PE}
          ;FOLD Parameters ;%{h}
          ;Params IlfProvider=kukaroboter.basistech.inlineforms.movement.spline; Kuka.IsGlobalPoint=False; Kuka.PointName=P500; Kuka.BlendingEnabled=False; Kuka.MoveDataPtpName=PDAT19; Kuka.VelocityPtp=100; Kuka.VelocityFieldEnabled=True; Kuka.ColDetectFieldEnabled=True; Kuka.CurrentCDSetIndex=0; Kuka.MovementParameterFieldEnabled=True; IlfCommand=SPTP
          ;ENDFOLD
          SPTP XP500 WITH $VEL_AXIS[1] = SVEL_JOINT(100.0), $TOOL = STOOL2(FP500), $BASE = SBASE(FP500.BASE_NO), $IPO_MODE = SIPO_MODE(FP500.IPO_FRAME), $LOAD = SLOAD(FP500.TOOL_NO), $ACC_AXIS[1] = SACC_JOINT(PPDAT19), $APO = SAPO_PTP(PPDAT19), $GEAR_JERK[1] = SGEAR_JERK(PPDAT19), $COLLMON_TOL_PRO[1] = USE_CM_PRO_VALUES(0)
          ;ENDFOLD
          ;FOLD Gripper SET [1]Gripper1 State=[1]ABIERTA Wait 0.2[s] Check with Strategy 1 ;%{PE}
          ;FOLD Parameters Parameters ;%{h}
          ;Params IlfProvider=GripperTech.GripperSet;setgripper=1;setstate=1;setcont=nocont;waittime=0.2;errorstrategy=1
          ;ENDFOLD
          GRPg_SetStateAndCheck(1, 1, 0.2, 1)
          ;ENDFOLD
      ENDIF
      IF eatPosition == 62 THEN
          ;FOLD SPTP P162 Vel=100 % PDAT1 Tool[1]:SMC Base[0] ;%{PE}
          ;FOLD Parameters ;%{h}
          ;Params IlfProvider=kukaroboter.basistech.inlineforms.movement.spline; Kuka.IsGlobalPoint=False; Kuka.PointName=P162; Kuka.BlendingEnabled=False; Kuka.MoveDataPtpName=PDAT1; Kuka.VelocityPtp=100; Kuka.VelocityFieldEnabled=True; Kuka.ColDetectFieldEnabled=True; Kuka.CurrentCDSetIndex=0; Kuka.MovementParameterFieldEnabled=True; IlfCommand=SPTP
          ;ENDFOLD
          SPTP XP162 WITH $VEL_AXIS[1] = SVEL_JOINT(100.0), $TOOL = STOOL2(FP162), $BASE = SBASE(FP162.BASE_NO), $IPO_MODE = SIPO_MODE(FP162.IPO_FRAME), $LOAD = SLOAD(FP162.TOOL_NO), $ACC_AXIS[1] = SACC_JOINT(PPDAT1), $APO = SAPO_PTP(PPDAT1), $GEAR_JERK[1] = SGEAR_JERK(PPDAT1), $COLLMON_TOL_PRO[1] = USE_CM_PRO_VALUES(0)
          ;ENDFOLD
          ;FOLD SLIN P262 Vel=0.1 m/s CPDAT32 Tool[1]:SMC Base[0] ;%{PE}
          ;FOLD Parameters ;%{h}
          ;Params IlfProvider=kukaroboter.basistech.inlineforms.movement.spline; Kuka.IsGlobalPoint=False; Kuka.PointName=P262; Kuka.BlendingEnabled=False; Kuka.MoveDataName=CPDAT32; Kuka.VelocityPath=0.1; Kuka.VelocityFieldEnabled=True; Kuka.ColDetectFieldEnabled=True; Kuka.CurrentCDSetIndex=0; Kuka.MovementParameterFieldEnabled=True; IlfCommand=SLIN
          ;ENDFOLD
          SLIN XP262 WITH $VEL = SVEL_CP(0.1, , LCPDAT32), $TOOL = STOOL2(FP262), $BASE = SBASE(FP262.BASE_NO), $IPO_MODE = SIPO_MODE(FP262.IPO_FRAME), $LOAD = SLOAD(FP262.TOOL_NO), $ACC = SACC_CP(LCPDAT32), $ORI_TYPE = SORI_TYP(LCPDAT32), $APO = SAPO(LCPDAT32), $JERK = SJERK(LCPDAT32), $COLLMON_TOL_PRO[1] = USE_CM_PRO_VALUES(0)
          ;ENDFOLD
          ;FOLD Gripper SET [1]Gripper1 State=[2]CERRADA Wait 0.2[s] Check with Strategy 1 ;%{PE}
          ;FOLD Parameters Parameters ;%{h}
          ;Params IlfProvider=GripperTech.GripperSet;setgripper=1;setstate=2;setcont=nocont;waittime=0.2;errorstrategy=1
          ;ENDFOLD
          GRPg_SetStateAndCheck(1, 2, 0.2, 1)
          ;ENDFOLDinitialPosition
          ;FOLD SLIN P162 Vel=0.1 m/s CPDAT33 Tool[1]:SMC Base[0] ;%{PE}
          ;FOLD Parameters ;%{h}s
          ;Params IlfProvider=kukaroboter.basistech.inlineforms.movement.spline; Kuka.IsGlobalPoint=False; Kuka.PointName=P162; Kuka.BlendingEnabled=False; Kuka.MoveDataName=CPDAT33; Kuka.VelocityPath=0.1; Kuka.VelocityFieldEnabled=True; Kuka.ColDetectFieldEnabled=True; Kuka.CurrentCDSetIndex=0; Kuka.MovementParameterFieldEnabled=True; IlfCommand=SLIN
          ;ENDFOLD
          SLIN XP162 WITH $VEL = SVEL_CP(0.1, , LCPDAT33), $TOOL = STOOL2(FP162), $BASE = SBASE(FP162.BASE_NO), $IPO_MODE = SIPO_MODE(FP162.IPO_FRAME), $LOAD = SLOAD(FP162.TOOL_NO), $ACC = SACC_CP(LCPDAT33), $ORI_TYPE = SORI_TYP(LCPDAT33), $APO = SAPO(LCPDAT33), $JERK = SJERK(LCPDAT33), $COLLMON_TOL_PRO[1] = USE_CM_PRO_VALUES(0)
          ;ENDFOLD
          ;FOLD SPTP P500 Vel=100 % PDAT19 Tool[1]:SMC Base[0] ;%{PE}
          ;FOLD Parameters ;%{h}
          ;Params IlfProvider=kukaroboter.basistech.inlineforms.movement.spline; Kuka.IsGlobalPoint=False; Kuka.PointName=P500; Kuka.BlendingEnabled=False; Kuka.MoveDataPtpName=PDAT19; Kuka.VelocityPtp=100; Kuka.VelocityFieldEnabled=True; Kuka.ColDetectFieldEnabled=True; Kuka.CurrentCDSetIndex=0; Kuka.MovementParameterFieldEnabled=True; IlfCommand=SPTP
          ;ENDFOLD
          SPTP XP500 WITH $VEL_AXIS[1] = SVEL_JOINT(100.0), $TOOL = STOOL2(FP500), $BASE = SBASE(FP500.BASE_NO), $IPO_MODE = SIPO_MODE(FP500.IPO_FRAME), $LOAD = SLOAD(FP500.TOOL_NO), $ACC_AXIS[1] = SACC_JOINT(PPDAT19), $APO = SAPO_PTP(PPDAT19), $GEAR_JERK[1] = SGEAR_JERK(PPDAT19), $COLLMON_TOL_PRO[1] = USE_CM_PRO_VALUES(0)
          ;ENDFOLD
          ;FOLD Gripper SET [1]Gripper1 State=[1]ABIERTA Wait 0.2[s] Check with Strategy 1 ;%{PE}
          ;FOLD Parameters Parameters ;%{h}
          ;Params IlfProvider=GripperTech.GripperSet;setgripper=1;setstate=1;setcont=nocont;waittime=0.2;errorstrategy=1
          ;ENDFOLD
          GRPg_SetStateAndCheck(1, 1, 0.2, 1)
          ;ENDFOLD
      ENDIF
      IF eatPosition == 63 THEN
          ;FOLD SPTP P163 Vel=100 % PDAT1 Tool[1]:SMC Base[0] ;%{PE}
          ;FOLD Parameters ;%{h}
          ;Params IlfProvider=kukaroboter.basistech.inlineforms.movement.spline; Kuka.IsGlobalPoint=False; Kuka.PointName=P163; Kuka.BlendingEnabled=False; Kuka.MoveDataPtpName=PDAT1; Kuka.VelocityPtp=100; Kuka.VelocityFieldEnabled=True; Kuka.ColDetectFieldEnabled=True; Kuka.CurrentCDSetIndex=0; Kuka.MovementParameterFieldEnabled=True; IlfCommand=SPTP
          ;ENDFOLD
          SPTP XP163 WITH $VEL_AXIS[1] = SVEL_JOINT(100.0), $TOOL = STOOL2(FP163), $BASE = SBASE(FP163.BASE_NO), $IPO_MODE = SIPO_MODE(FP163.IPO_FRAME), $LOAD = SLOAD(FP163.TOOL_NO), $ACC_AXIS[1] = SACC_JOINT(PPDAT1), $APO = SAPO_PTP(PPDAT1), $GEAR_JERK[1] = SGEAR_JERK(PPDAT1), $COLLMON_TOL_PRO[1] = USE_CM_PRO_VALUES(0)
          ;ENDFOLD
          ;FOLD SLIN P263 Vel=0.1 m/s CPDAT32 Tool[1]:SMC Base[0] ;%{PE}
          ;FOLD Parameters ;%{h}
          ;Params IlfProvider=kukaroboter.basistech.inlineforms.movement.spline; Kuka.IsGlobalPoint=False; Kuka.PointName=P263; Kuka.BlendingEnabled=False; Kuka.MoveDataName=CPDAT32; Kuka.VelocityPath=0.1; Kuka.VelocityFieldEnabled=True; Kuka.ColDetectFieldEnabled=True; Kuka.CurrentCDSetIndex=0; Kuka.MovementParameterFieldEnabled=True; IlfCommand=SLIN
          ;ENDFOLD
          SLIN XP263 WITH $VEL = SVEL_CP(0.1, , LCPDAT32), $TOOL = STOOL2(FP263), $BASE = SBASE(FP263.BASE_NO), $IPO_MODE = SIPO_MODE(FP263.IPO_FRAME), $LOAD = SLOAD(FP263.TOOL_NO), $ACC = SACC_CP(LCPDAT32), $ORI_TYPE = SORI_TYP(LCPDAT32), $APO = SAPO(LCPDAT32), $JERK = SJERK(LCPDAT32), $COLLMON_TOL_PRO[1] = USE_CM_PRO_VALUES(0)
          ;ENDFOLD
          ;FOLD Gripper SET [1]Gripper1 State=[2]CERRADA Wait 0.2[s] Check with Strategy 1 ;%{PE}
          ;FOLD Parameters Parameters ;%{h}
          ;Params IlfProvider=GripperTech.GripperSet;setgripper=1;setstate=2;setcont=nocont;waittime=0.2;errorstrategy=1
          ;ENDFOLD
          GRPg_SetStateAndCheck(1, 2, 0.2, 1)
          ;ENDFOLDinitialPosition
          ;FOLD SLIN P163 Vel=0.1 m/s CPDAT33 Tool[1]:SMC Base[0] ;%{PE}
          ;FOLD Parameters ;%{h}s
          ;Params IlfProvider=kukaroboter.basistech.inlineforms.movement.spline; Kuka.IsGlobalPoint=False; Kuka.PointName=P163; Kuka.BlendingEnabled=False; Kuka.MoveDataName=CPDAT33; Kuka.VelocityPath=0.1; Kuka.VelocityFieldEnabled=True; Kuka.ColDetectFieldEnabled=True; Kuka.CurrentCDSetIndex=0; Kuka.MovementParameterFieldEnabled=True; IlfCommand=SLIN
          ;ENDFOLD
          SLIN XP163 WITH $VEL = SVEL_CP(0.1, , LCPDAT33), $TOOL = STOOL2(FP163), $BASE = SBASE(FP163.BASE_NO), $IPO_MODE = SIPO_MODE(FP163.IPO_FRAME), $LOAD = SLOAD(FP163.TOOL_NO), $ACC = SACC_CP(LCPDAT33), $ORI_TYPE = SORI_TYP(LCPDAT33), $APO = SAPO(LCPDAT33), $JERK = SJERK(LCPDAT33), $COLLMON_TOL_PRO[1] = USE_CM_PRO_VALUES(0)
          ;ENDFOLD
          ;FOLD SPTP P500 Vel=100 % PDAT19 Tool[1]:SMC Base[0] ;%{PE}
          ;FOLD Parameters ;%{h}
          ;Params IlfProvider=kukaroboter.basistech.inlineforms.movement.spline; Kuka.IsGlobalPoint=False; Kuka.PointName=P500; Kuka.BlendingEnabled=False; Kuka.MoveDataPtpName=PDAT19; Kuka.VelocityPtp=100; Kuka.VelocityFieldEnabled=True; Kuka.ColDetectFieldEnabled=True; Kuka.CurrentCDSetIndex=0; Kuka.MovementParameterFieldEnabled=True; IlfCommand=SPTP
          ;ENDFOLD
          SPTP XP500 WITH $VEL_AXIS[1] = SVEL_JOINT(100.0), $TOOL = STOOL2(FP500), $BASE = SBASE(FP500.BASE_NO), $IPO_MODE = SIPO_MODE(FP500.IPO_FRAME), $LOAD = SLOAD(FP500.TOOL_NO), $ACC_AXIS[1] = SACC_JOINT(PPDAT19), $APO = SAPO_PTP(PPDAT19), $GEAR_JERK[1] = SGEAR_JERK(PPDAT19), $COLLMON_TOL_PRO[1] = USE_CM_PRO_VALUES(0)
          ;ENDFOLD
          ;FOLD Gripper SET [1]Gripper1 State=[1]ABIERTA Wait 0.2[s] Check with Strategy 1 ;%{PE}
          ;FOLD Parameters Parameters ;%{h}
          ;Params IlfProvider=GripperTech.GripperSet;setgripper=1;setstate=1;setcont=nocont;waittime=0.2;errorstrategy=1
          ;ENDFOLD
          GRPg_SetStateAndCheck(1, 1, 0.2, 1)
          ;ENDFOLD
      ENDIF
      IF eatPosition == 64 THEN
          ;FOLD SPTP P164 Vel=100 % PDAT1 Tool[1]:SMC Base[0] ;%{PE}
          ;FOLD Parameters ;%{h}
          ;Params IlfProvider=kukaroboter.basistech.inlineforms.movement.spline; Kuka.IsGlobalPoint=False; Kuka.PointName=P164; Kuka.BlendingEnabled=False; Kuka.MoveDataPtpName=PDAT1; Kuka.VelocityPtp=100; Kuka.VelocityFieldEnabled=True; Kuka.ColDetectFieldEnabled=True; Kuka.CurrentCDSetIndex=0; Kuka.MovementParameterFieldEnabled=True; IlfCommand=SPTP
          ;ENDFOLD
          SPTP XP164 WITH $VEL_AXIS[1] = SVEL_JOINT(100.0), $TOOL = STOOL2(FP164), $BASE = SBASE(FP164.BASE_NO), $IPO_MODE = SIPO_MODE(FP164.IPO_FRAME), $LOAD = SLOAD(FP164.TOOL_NO), $ACC_AXIS[1] = SACC_JOINT(PPDAT1), $APO = SAPO_PTP(PPDAT1), $GEAR_JERK[1] = SGEAR_JERK(PPDAT1), $COLLMON_TOL_PRO[1] = USE_CM_PRO_VALUES(0)
          ;ENDFOLD
          ;FOLD SLIN P264 Vel=0.1 m/s CPDAT32 Tool[1]:SMC Base[0] ;%{PE}
          ;FOLD Parameters ;%{h}
          ;Params IlfProvider=kukaroboter.basistech.inlineforms.movement.spline; Kuka.IsGlobalPoint=False; Kuka.PointName=P264; Kuka.BlendingEnabled=False; Kuka.MoveDataName=CPDAT32; Kuka.VelocityPath=0.1; Kuka.VelocityFieldEnabled=True; Kuka.ColDetectFieldEnabled=True; Kuka.CurrentCDSetIndex=0; Kuka.MovementParameterFieldEnabled=True; IlfCommand=SLIN
          ;ENDFOLD
          SLIN XP264 WITH $VEL = SVEL_CP(0.1, , LCPDAT32), $TOOL = STOOL2(FP264), $BASE = SBASE(FP264.BASE_NO), $IPO_MODE = SIPO_MODE(FP264.IPO_FRAME), $LOAD = SLOAD(FP264.TOOL_NO), $ACC = SACC_CP(LCPDAT32), $ORI_TYPE = SORI_TYP(LCPDAT32), $APO = SAPO(LCPDAT32), $JERK = SJERK(LCPDAT32), $COLLMON_TOL_PRO[1] = USE_CM_PRO_VALUES(0)
          ;ENDFOLD
          ;FOLD Gripper SET [1]Gripper1 State=[2]CERRADA Wait 0.2[s] Check with Strategy 1 ;%{PE}
          ;FOLD Parameters Parameters ;%{h}
          ;Params IlfProvider=GripperTech.GripperSet;setgripper=1;setstate=2;setcont=nocont;waittime=0.2;errorstrategy=1
          ;ENDFOLD
          GRPg_SetStateAndCheck(1, 2, 0.2, 1)
          ;ENDFOLDinitialPosition
          ;FOLD SLIN P164 Vel=0.1 m/s CPDAT33 Tool[1]:SMC Base[0] ;%{PE}
          ;FOLD Parameters ;%{h}s
          ;Params IlfProvider=kukaroboter.basistech.inlineforms.movement.spline; Kuka.IsGlobalPoint=False; Kuka.PointName=P164; Kuka.BlendingEnabled=False; Kuka.MoveDataName=CPDAT33; Kuka.VelocityPath=0.1; Kuka.VelocityFieldEnabled=True; Kuka.ColDetectFieldEnabled=True; Kuka.CurrentCDSetIndex=0; Kuka.MovementParameterFieldEnabled=True; IlfCommand=SLIN
          ;ENDFOLD
          SLIN XP164 WITH $VEL = SVEL_CP(0.1, , LCPDAT33), $TOOL = STOOL2(FP164), $BASE = SBASE(FP164.BASE_NO), $IPO_MODE = SIPO_MODE(FP164.IPO_FRAME), $LOAD = SLOAD(FP164.TOOL_NO), $ACC = SACC_CP(LCPDAT33), $ORI_TYPE = SORI_TYP(LCPDAT33), $APO = SAPO(LCPDAT33), $JERK = SJERK(LCPDAT33), $COLLMON_TOL_PRO[1] = USE_CM_PRO_VALUES(0)
          ;ENDFOLD
          ;FOLD SPTP P500 Vel=100 % PDAT19 Tool[1]:SMC Base[0] ;%{PE}
          ;FOLD Parameters ;%{h}
          ;Params IlfProvider=kukaroboter.basistech.inlineforms.movement.spline; Kuka.IsGlobalPoint=False; Kuka.PointName=P500; Kuka.BlendingEnabled=False; Kuka.MoveDataPtpName=PDAT19; Kuka.VelocityPtp=100; Kuka.VelocityFieldEnabled=True; Kuka.ColDetectFieldEnabled=True; Kuka.CurrentCDSetIndex=0; Kuka.MovementParameterFieldEnabled=True; IlfCommand=SPTP
          ;ENDFOLD
          SPTP XP500 WITH $VEL_AXIS[1] = SVEL_JOINT(100.0), $TOOL = STOOL2(FP500), $BASE = SBASE(FP500.BASE_NO), $IPO_MODE = SIPO_MODE(FP500.IPO_FRAME), $LOAD = SLOAD(FP500.TOOL_NO), $ACC_AXIS[1] = SACC_JOINT(PPDAT19), $APO = SAPO_PTP(PPDAT19), $GEAR_JERK[1] = SGEAR_JERK(PPDAT19), $COLLMON_TOL_PRO[1] = USE_CM_PRO_VALUES(0)
          ;ENDFOLD
          ;FOLD Gripper SET [1]Gripper1 State=[1]ABIERTA Wait 0.2[s] Check with Strategy 1 ;%{PE}
          ;FOLD Parameters Parameters ;%{h}
          ;Params IlfProvider=GripperTech.GripperSet;setgripper=1;setstate=1;setcont=nocont;waittime=0.2;errorstrategy=1
          ;ENDFOLD
          GRPg_SetStateAndCheck(1, 1, 0.2, 1)
          ;ENDFOLD
      ENDIF

      IF initialPosition == 1 THEN
        ;FOLD SPTP P101 Vel=100 % PDAT1 Tool[1]:SMC Base[0] ;%{PE}
        ;FOLD Parameters ;%{h}
        ;Params IlfProvider=kukaroboter.basistech.inlineforms.movement.spline; Kuka.IsGlobalPoint=False; Kuka.PointName=P101; Kuka.BlendingEnabled=False; Kuka.MoveDataPtpName=PDAT1; Kuka.VelocityPtp=100; Kuka.VelocityFieldEnabled=True; Kuka.ColDetectFieldEnabled=True; Kuka.CurrentCDSetIndex=0; Kuka.MovementParameterFieldEnabled=True; IlfCommand=SPTP
        ;ENDFOLD
        SPTP XP101 WITH $VEL_AXIS[1] = SVEL_JOINT(100.0), $TOOL = STOOL2(FP101), $BASE = SBASE(FP101.BASE_NO), $IPO_MODE = SIPO_MODE(FP101.IPO_FRAME), $LOAD = SLOAD(FP101.TOOL_NO), $ACC_AXIS[1] = SACC_JOINT(PPDAT1), $APO = SAPO_PTP(PPDAT1), $GEAR_JERK[1] = SGEAR_JERK(PPDAT1), $COLLMON_TOL_PRO[1] = USE_CM_PRO_VALUES(0)
        ;ENDFOLD
        ;FOLD SLIN P201 Vel=0.1 m/s CPDAT27 Tool[1]:SMC Base[0] ;%{PE}
        ;FOLD Parameters ;%{h}
        ;Params IlfProvider=kukaroboter.basistech.inlineforms.movement.spline; Kuka.IsGlobalPoint=False; Kuka.PointName=P201; Kuka.BlendingEnabled=False; Kuka.MoveDataName=CPDAT27; Kuka.VelocityPath=0.1; Kuka.VelocityFieldEnabled=True; Kuka.ColDetectFieldEnabled=True; Kuka.CurrentCDSetIndex=0; Kuka.MovementParameterFieldEnabled=True; IlfCommand=SLIN
        ;ENDFOLD
        SLIN XP201 WITH $VEL = SVEL_CP(0.1, , LCPDAT27), $TOOL = STOOL2(FP201), $BASE = SBASE(FP201.BASE_NO), $IPO_MODE = SIPO_MODE(FP201.IPO_FRAME), $LOAD = SLOAD(FP201.TOOL_NO), $ACC = SACC_CP(LCPDAT27), $ORI_TYPE = SORI_TYP(LCPDAT27), $APO = SAPO(LCPDAT27), $JERK = SJERK(LCPDAT27), $COLLMON_TOL_PRO[1] = USE_CM_PRO_VALUES(0)
        ;ENDFOLD
        ;FOLD Gripper SET [1]Gripper1 State=[2]CERRADA Wait 0.2[s] Check with Strategy 1 ;%{PE}
        ;FOLD Parameters Parameters ;%{h}
        ;Params IlfProvider=GripperTech.GripperSet;setgripper=1;setstate=2;setcont=nocont;waittime=0.2;errorstrategy=1
        ;ENDFOLD
        GRPg_SetStateAndCheck(1, 2, 0.2, 1)
        ;ENDFOLD
        ;FOLD SLIN P101 Vel=0.1 m/s CPDAT28 Tool[1]:SMC Base[0] ;%{PE}
        ;FOLD Parameters ;%{h}
        ;Params IlfProvider=kukaroboter.basistech.inlineforms.movement.spline; Kuka.IsGlobalPoint=False; Kuka.PointName=P101; Kuka.BlendingEnabled=False; Kuka.MoveDataName=CPDAT28; Kuka.VelocityPath=0.1; Kuka.VelocityFieldEnabled=True; Kuka.ColDetectFieldEnabled=True; Kuka.CurrentCDSetIndex=0; Kuka.MovementParameterFieldEnabled=True; IlfCommand=SLIN
        ;ENDFOLD
        SLIN XP101 WITH $VEL = SVEL_CP(0.1, , LCPDAT28), $TOOL = STOOL2(FP101), $BASE = SBASE(FP101.BASE_NO), $IPO_MODE = SIPO_MODE(FP101.IPO_FRAME), $LOAD = SLOAD(FP101.TOOL_NO), $ACC = SACC_CP(LCPDAT28), $ORI_TYPE = SORI_TYP(LCPDAT28), $APO = SAPO(LCPDAT28), $JERK = SJERK(LCPDAT28), $COLLMON_TOL_PRO[1] = USE_CM_PRO_VALUES(0)
        ;ENDFOLD
      ENDIF

      IF initialPosition == 2 THEN
        ;FOLD SPTP P102 Vel=100 % PDAT1 Tool[1]:SMC Base[0] ;%{PE}
        ;FOLD Parameters ;%{h}
        ;Params IlfProvider=kukaroboter.basistech.inlineforms.movement.spline; Kuka.IsGlobalPoint=False; Kuka.PointName=P102; Kuka.BlendingEnabled=False; Kuka.MoveDataPtpName=PDAT1; Kuka.VelocityPtp=100; Kuka.VelocityFieldEnabled=True; Kuka.ColDetectFieldEnabled=True; Kuka.CurrentCDSetIndex=0; Kuka.MovementParameterFieldEnabled=True; IlfCommand=SPTP
        ;ENDFOLD
        SPTP XP102 WITH $VEL_AXIS[1] = SVEL_JOINT(100.0), $TOOL = STOOL2(FP102), $BASE = SBASE(FP102.BASE_NO), $IPO_MODE = SIPO_MODE(FP102.IPO_FRAME), $LOAD = SLOAD(FP102.TOOL_NO), $ACC_AXIS[1] = SACC_JOINT(PPDAT1), $APO = SAPO_PTP(PPDAT1), $GEAR_JERK[1] = SGEAR_JERK(PPDAT1), $COLLMON_TOL_PRO[1] = USE_CM_PRO_VALUES(0)
        ;ENDFOLD
        ;FOLD SLIN P202 Vel=0.1 m/s CPDAT27 Tool[1]:SMC Base[0] ;%{PE}
        ;FOLD Parameters ;%{h}
        ;Params IlfProvider=kukaroboter.basistech.inlineforms.movement.spline; Kuka.IsGlobalPoint=False; Kuka.PointName=P202; Kuka.BlendingEnabled=False; Kuka.MoveDataName=CPDAT27; Kuka.VelocityPath=0.1; Kuka.VelocityFieldEnabled=True; Kuka.ColDetectFieldEnabled=True; Kuka.CurrentCDSetIndex=0; Kuka.MovementParameterFieldEnabled=True; IlfCommand=SLIN
        ;ENDFOLD
        SLIN XP202 WITH $VEL = SVEL_CP(0.1, , LCPDAT27), $TOOL = STOOL2(FP202), $BASE = SBASE(FP202.BASE_NO), $IPO_MODE = SIPO_MODE(FP202.IPO_FRAME), $LOAD = SLOAD(FP202.TOOL_NO), $ACC = SACC_CP(LCPDAT27), $ORI_TYPE = SORI_TYP(LCPDAT27), $APO = SAPO(LCPDAT27), $JERK = SJERK(LCPDAT27), $COLLMON_TOL_PRO[1] = USE_CM_PRO_VALUES(0)
        ;ENDFOLD
        ;FOLD Gripper SET [1]Gripper1 State=[2]CERRADA Wait 0.2[s] Check with Strategy 1 ;%{PE}
        ;FOLD Parameters Parameters ;%{h}
        ;Params IlfProvider=GripperTech.GripperSet;setgripper=1;setstate=2;setcont=nocont;waittime=0.2;errorstrategy=1
        ;ENDFOLD
        GRPg_SetStateAndCheck(1, 2, 0.2, 1)
        ;ENDFOLD
        ;FOLD SLIN P102 Vel=0.1 m/s CPDAT28 Tool[1]:SMC Base[0] ;%{PE}
        ;FOLD Parameters ;%{h}
        ;Params IlfProvider=kukaroboter.basistech.inlineforms.movement.spline; Kuka.IsGlobalPoint=False; Kuka.PointName=P102; Kuka.BlendingEnabled=False; Kuka.MoveDataName=CPDAT28; Kuka.VelocityPath=0.1; Kuka.VelocityFieldEnabled=True; Kuka.ColDetectFieldEnabled=True; Kuka.CurrentCDSetIndex=0; Kuka.MovementParameterFieldEnabled=True; IlfCommand=SLIN
        ;ENDFOLD
        SLIN XP102 WITH $VEL = SVEL_CP(0.1, , LCPDAT28), $TOOL = STOOL2(FP102), $BASE = SBASE(FP102.BASE_NO), $IPO_MODE = SIPO_MODE(FP102.IPO_FRAME), $LOAD = SLOAD(FP102.TOOL_NO), $ACC = SACC_CP(LCPDAT28), $ORI_TYPE = SORI_TYP(LCPDAT28), $APO = SAPO(LCPDAT28), $JERK = SJERK(LCPDAT28), $COLLMON_TOL_PRO[1] = USE_CM_PRO_VALUES(0)
        ;ENDFOLD
      ENDIF

      IF initialPosition == 3 THEN
        ;FOLD SPTP P103 Vel=100 % PDAT1 Tool[1]:SMC Base[0] ;%{PE}
        ;FOLD Parameters ;%{h}
        ;Params IlfProvider=kukaroboter.basistech.inlineforms.movement.spline; Kuka.IsGlobalPoint=False; Kuka.PointName=P103; Kuka.BlendingEnabled=False; Kuka.MoveDataPtpName=PDAT1; Kuka.VelocityPtp=100; Kuka.VelocityFieldEnabled=True; Kuka.ColDetectFieldEnabled=True; Kuka.CurrentCDSetIndex=0; Kuka.MovementParameterFieldEnabled=True; IlfCommand=SPTP
        ;ENDFOLD
        SPTP XP103 WITH $VEL_AXIS[1] = SVEL_JOINT(100.0), $TOOL = STOOL2(FP103), $BASE = SBASE(FP103.BASE_NO), $IPO_MODE = SIPO_MODE(FP103.IPO_FRAME), $LOAD = SLOAD(FP103.TOOL_NO), $ACC_AXIS[1] = SACC_JOINT(PPDAT1), $APO = SAPO_PTP(PPDAT1), $GEAR_JERK[1] = SGEAR_JERK(PPDAT1), $COLLMON_TOL_PRO[1] = USE_CM_PRO_VALUES(0)
        ;ENDFOLD
        ;FOLD SLIN P203 Vel=0.1 m/s CPDAT27 Tool[1]:SMC Base[0] ;%{PE}
        ;FOLD Parameters ;%{h}
        ;Params IlfProvider=kukaroboter.basistech.inlineforms.movement.spline; Kuka.IsGlobalPoint=False; Kuka.PointName=P203; Kuka.BlendingEnabled=False; Kuka.MoveDataName=CPDAT27; Kuka.VelocityPath=0.1; Kuka.VelocityFieldEnabled=True; Kuka.ColDetectFieldEnabled=True; Kuka.CurrentCDSetIndex=0; Kuka.MovementParameterFieldEnabled=True; IlfCommand=SLIN
        ;ENDFOLD
        SLIN XP203 WITH $VEL = SVEL_CP(0.1, , LCPDAT27), $TOOL = STOOL2(FP203), $BASE = SBASE(FP203.BASE_NO), $IPO_MODE = SIPO_MODE(FP203.IPO_FRAME), $LOAD = SLOAD(FP203.TOOL_NO), $ACC = SACC_CP(LCPDAT27), $ORI_TYPE = SORI_TYP(LCPDAT27), $APO = SAPO(LCPDAT27), $JERK = SJERK(LCPDAT27), $COLLMON_TOL_PRO[1] = USE_CM_PRO_VALUES(0)
        ;ENDFOLD
        ;FOLD Gripper SET [1]Gripper1 State=[2]CERRADA Wait 0.2[s] Check with Strategy 1 ;%{PE}
        ;FOLD Parameters Parameters ;%{h}
        ;Params IlfProvider=GripperTech.GripperSet;setgripper=1;setstate=2;setcont=nocont;waittime=0.2;errorstrategy=1
        ;ENDFOLD
        GRPg_SetStateAndCheck(1, 2, 0.2, 1)
        ;ENDFOLD
        ;FOLD SLIN P103 Vel=0.1 m/s CPDAT28 Tool[1]:SMC Base[0] ;%{PE}
        ;FOLD Parameters ;%{h}
        ;Params IlfProvider=kukaroboter.basistech.inlineforms.movement.spline; Kuka.IsGlobalPoint=False; Kuka.PointName=P103; Kuka.BlendingEnabled=False; Kuka.MoveDataName=CPDAT28; Kuka.VelocityPath=0.1; Kuka.VelocityFieldEnabled=True; Kuka.ColDetectFieldEnabled=True; Kuka.CurrentCDSetIndex=0; Kuka.MovementParameterFieldEnabled=True; IlfCommand=SLIN
        ;ENDFOLD
        SLIN XP103 WITH $VEL = SVEL_CP(0.1, , LCPDAT28), $TOOL = STOOL2(FP103), $BASE = SBASE(FP103.BASE_NO), $IPO_MODE = SIPO_MODE(FP103.IPO_FRAME), $LOAD = SLOAD(FP103.TOOL_NO), $ACC = SACC_CP(LCPDAT28), $ORI_TYPE = SORI_TYP(LCPDAT28), $APO = SAPO(LCPDAT28), $JERK = SJERK(LCPDAT28), $COLLMON_TOL_PRO[1] = USE_CM_PRO_VALUES(0)
        ;ENDFOLD
      ENDIF

      IF initialPosition == 4 THEN
        ;FOLD SPTP P104 Vel=100 % PDAT1 Tool[1]:SMC Base[0] ;%{PE}
        ;FOLD Parameters ;%{h}
        ;Params IlfProvider=kukaroboter.basistech.inlineforms.movement.spline; Kuka.IsGlobalPoint=False; Kuka.PointName=P104; Kuka.BlendingEnabled=False; Kuka.MoveDataPtpName=PDAT1; Kuka.VelocityPtp=100; Kuka.VelocityFieldEnabled=True; Kuka.ColDetectFieldEnabled=True; Kuka.CurrentCDSetIndex=0; Kuka.MovementParameterFieldEnabled=True; IlfCommand=SPTP
        ;ENDFOLD
        SPTP XP104 WITH $VEL_AXIS[1] = SVEL_JOINT(100.0), $TOOL = STOOL2(FP104), $BASE = SBASE(FP104.BASE_NO), $IPO_MODE = SIPO_MODE(FP104.IPO_FRAME), $LOAD = SLOAD(FP104.TOOL_NO), $ACC_AXIS[1] = SACC_JOINT(PPDAT1), $APO = SAPO_PTP(PPDAT1), $GEAR_JERK[1] = SGEAR_JERK(PPDAT1), $COLLMON_TOL_PRO[1] = USE_CM_PRO_VALUES(0)
        ;ENDFOLD
        ;FOLD SLIN P204 Vel=0.1 m/s CPDAT27 Tool[1]:SMC Base[0] ;%{PE}
        ;FOLD Parameters ;%{h}
        ;Params IlfProvider=kukaroboter.basistech.inlineforms.movement.spline; Kuka.IsGlobalPoint=False; Kuka.PointName=P204; Kuka.BlendingEnabled=False; Kuka.MoveDataName=CPDAT27; Kuka.VelocityPath=0.1; Kuka.VelocityFieldEnabled=True; Kuka.ColDetectFieldEnabled=True; Kuka.CurrentCDSetIndex=0; Kuka.MovementParameterFieldEnabled=True; IlfCommand=SLIN
        ;ENDFOLD
        SLIN XP204 WITH $VEL = SVEL_CP(0.1, , LCPDAT27), $TOOL = STOOL2(FP204), $BASE = SBASE(FP204.BASE_NO), $IPO_MODE = SIPO_MODE(FP204.IPO_FRAME), $LOAD = SLOAD(FP204.TOOL_NO), $ACC = SACC_CP(LCPDAT27), $ORI_TYPE = SORI_TYP(LCPDAT27), $APO = SAPO(LCPDAT27), $JERK = SJERK(LCPDAT27), $COLLMON_TOL_PRO[1] = USE_CM_PRO_VALUES(0)
        ;ENDFOLD
        ;FOLD Gripper SET [1]Gripper1 State=[2]CERRADA Wait 0.2[s] Check with Strategy 1 ;%{PE}
        ;FOLD Parameters Parameters ;%{h}
        ;Params IlfProvider=GripperTech.GripperSet;setgripper=1;setstate=2;setcont=nocont;waittime=0.2;errorstrategy=1
        ;ENDFOLD
        GRPg_SetStateAndCheck(1, 2, 0.2, 1)
        ;ENDFOLD
        ;FOLD SLIN P104 Vel=0.1 m/s CPDAT28 Tool[1]:SMC Base[0] ;%{PE}
        ;FOLD Parameters ;%{h}
        ;Params IlfProvider=kukaroboter.basistech.inlineforms.movement.spline; Kuka.IsGlobalPoint=False; Kuka.PointName=P104; Kuka.BlendingEnabled=False; Kuka.MoveDataName=CPDAT28; Kuka.VelocityPath=0.1; Kuka.VelocityFieldEnabled=True; Kuka.ColDetectFieldEnabled=True; Kuka.CurrentCDSetIndex=0; Kuka.MovementParameterFieldEnabled=True; IlfCommand=SLIN
        ;ENDFOLD
        SLIN XP104 WITH $VEL = SVEL_CP(0.1, , LCPDAT28), $TOOL = STOOL2(FP104), $BASE = SBASE(FP104.BASE_NO), $IPO_MODE = SIPO_MODE(FP104.IPO_FRAME), $LOAD = SLOAD(FP104.TOOL_NO), $ACC = SACC_CP(LCPDAT28), $ORI_TYPE = SORI_TYP(LCPDAT28), $APO = SAPO(LCPDAT28), $JERK = SJERK(LCPDAT28), $COLLMON_TOL_PRO[1] = USE_CM_PRO_VALUES(0)
        ;ENDFOLD
      ENDIF

      IF initialPosition == 5 THEN
        ;FOLD SPTP P105 Vel=100 % PDAT1 Tool[1]:SMC Base[0] ;%{PE}
        ;FOLD Parameters ;%{h}
        ;Params IlfProvider=kukaroboter.basistech.inlineforms.movement.spline; Kuka.IsGlobalPoint=False; Kuka.PointName=P105; Kuka.BlendingEnabled=False; Kuka.MoveDataPtpName=PDAT1; Kuka.VelocityPtp=100; Kuka.VelocityFieldEnabled=True; Kuka.ColDetectFieldEnabled=True; Kuka.CurrentCDSetIndex=0; Kuka.MovementParameterFieldEnabled=True; IlfCommand=SPTP
        ;ENDFOLD
        SPTP XP105 WITH $VEL_AXIS[1] = SVEL_JOINT(100.0), $TOOL = STOOL2(FP105), $BASE = SBASE(FP105.BASE_NO), $IPO_MODE = SIPO_MODE(FP105.IPO_FRAME), $LOAD = SLOAD(FP105.TOOL_NO), $ACC_AXIS[1] = SACC_JOINT(PPDAT1), $APO = SAPO_PTP(PPDAT1), $GEAR_JERK[1] = SGEAR_JERK(PPDAT1), $COLLMON_TOL_PRO[1] = USE_CM_PRO_VALUES(0)
        ;ENDFOLD
        ;FOLD SLIN P205 Vel=0.1 m/s CPDAT27 Tool[1]:SMC Base[0] ;%{PE}
        ;FOLD Parameters ;%{h}
        ;Params IlfProvider=kukaroboter.basistech.inlineforms.movement.spline; Kuka.IsGlobalPoint=False; Kuka.PointName=P205; Kuka.BlendingEnabled=False; Kuka.MoveDataName=CPDAT27; Kuka.VelocityPath=0.1; Kuka.VelocityFieldEnabled=True; Kuka.ColDetectFieldEnabled=True; Kuka.CurrentCDSetIndex=0; Kuka.MovementParameterFieldEnabled=True; IlfCommand=SLIN
        ;ENDFOLD
        SLIN XP205 WITH $VEL = SVEL_CP(0.1, , LCPDAT27), $TOOL = STOOL2(FP205), $BASE = SBASE(FP205.BASE_NO), $IPO_MODE = SIPO_MODE(FP205.IPO_FRAME), $LOAD = SLOAD(FP205.TOOL_NO), $ACC = SACC_CP(LCPDAT27), $ORI_TYPE = SORI_TYP(LCPDAT27), $APO = SAPO(LCPDAT27), $JERK = SJERK(LCPDAT27), $COLLMON_TOL_PRO[1] = USE_CM_PRO_VALUES(0)
        ;ENDFOLD
        ;FOLD Gripper SET [1]Gripper1 State=[2]CERRADA Wait 0.2[s] Check with Strategy 1 ;%{PE}
        ;FOLD Parameters Parameters ;%{h}
        ;Params IlfProvider=GripperTech.GripperSet;setgripper=1;setstate=2;setcont=nocont;waittime=0.2;errorstrategy=1
        ;ENDFOLD
        GRPg_SetStateAndCheck(1, 2, 0.2, 1)
        ;ENDFOLD
        ;FOLD SLIN P105 Vel=0.1 m/s CPDAT28 Tool[1]:SMC Base[0] ;%{PE}
        ;FOLD Parameters ;%{h}
        ;Params IlfProvider=kukaroboter.basistech.inlineforms.movement.spline; Kuka.IsGlobalPoint=False; Kuka.PointName=P105; Kuka.BlendingEnabled=False; Kuka.MoveDataName=CPDAT28; Kuka.VelocityPath=0.1; Kuka.VelocityFieldEnabled=True; Kuka.ColDetectFieldEnabled=True; Kuka.CurrentCDSetIndex=0; Kuka.MovementParameterFieldEnabled=True; IlfCommand=SLIN
        ;ENDFOLD
        SLIN XP105 WITH $VEL = SVEL_CP(0.1, , LCPDAT28), $TOOL = STOOL2(FP105), $BASE = SBASE(FP105.BASE_NO), $IPO_MODE = SIPO_MODE(FP105.IPO_FRAME), $LOAD = SLOAD(FP105.TOOL_NO), $ACC = SACC_CP(LCPDAT28), $ORI_TYPE = SORI_TYP(LCPDAT28), $APO = SAPO(LCPDAT28), $JERK = SJERK(LCPDAT28), $COLLMON_TOL_PRO[1] = USE_CM_PRO_VALUES(0)
        ;ENDFOLD
      ENDIF

      IF initialPosition == 6 THEN
        ;FOLD SPTP P106 Vel=100 % PDAT1 Tool[1]:SMC Base[0] ;%{PE}
        ;FOLD Parameters ;%{h}
        ;Params IlfProvider=kukaroboter.basistech.inlineforms.movement.spline; Kuka.IsGlobalPoint=False; Kuka.PointName=P106; Kuka.BlendingEnabled=False; Kuka.MoveDataPtpName=PDAT1; Kuka.VelocityPtp=100; Kuka.VelocityFieldEnabled=True; Kuka.ColDetectFieldEnabled=True; Kuka.CurrentCDSetIndex=0; Kuka.MovementParameterFieldEnabled=True; IlfCommand=SPTP
        ;ENDFOLD
        SPTP XP106 WITH $VEL_AXIS[1] = SVEL_JOINT(100.0), $TOOL = STOOL2(FP106), $BASE = SBASE(FP106.BASE_NO), $IPO_MODE = SIPO_MODE(FP106.IPO_FRAME), $LOAD = SLOAD(FP106.TOOL_NO), $ACC_AXIS[1] = SACC_JOINT(PPDAT1), $APO = SAPO_PTP(PPDAT1), $GEAR_JERK[1] = SGEAR_JERK(PPDAT1), $COLLMON_TOL_PRO[1] = USE_CM_PRO_VALUES(0)
        ;ENDFOLD
        ;FOLD SLIN P206 Vel=0.1 m/s CPDAT27 Tool[1]:SMC Base[0] ;%{PE}
        ;FOLD Parameters ;%{h}
        ;Params IlfProvider=kukaroboter.basistech.inlineforms.movement.spline; Kuka.IsGlobalPoint=False; Kuka.PointName=P206; Kuka.BlendingEnabled=False; Kuka.MoveDataName=CPDAT27; Kuka.VelocityPath=0.1; Kuka.VelocityFieldEnabled=True; Kuka.ColDetectFieldEnabled=True; Kuka.CurrentCDSetIndex=0; Kuka.MovementParameterFieldEnabled=True; IlfCommand=SLIN
        ;ENDFOLD
        SLIN XP206 WITH $VEL = SVEL_CP(0.1, , LCPDAT27), $TOOL = STOOL2(FP206), $BASE = SBASE(FP206.BASE_NO), $IPO_MODE = SIPO_MODE(FP206.IPO_FRAME), $LOAD = SLOAD(FP206.TOOL_NO), $ACC = SACC_CP(LCPDAT27), $ORI_TYPE = SORI_TYP(LCPDAT27), $APO = SAPO(LCPDAT27), $JERK = SJERK(LCPDAT27), $COLLMON_TOL_PRO[1] = USE_CM_PRO_VALUES(0)
        ;ENDFOLD
        ;FOLD Gripper SET [1]Gripper1 State=[2]CERRADA Wait 0.2[s] Check with Strategy 1 ;%{PE}
        ;FOLD Parameters Parameters ;%{h}
        ;Params IlfProvider=GripperTech.GripperSet;setgripper=1;setstate=2;setcont=nocont;waittime=0.2;errorstrategy=1
        ;ENDFOLD
        GRPg_SetStateAndCheck(1, 2, 0.2, 1)
        ;ENDFOLD
        ;FOLD SLIN P106 Vel=0.1 m/s CPDAT28 Tool[1]:SMC Base[0] ;%{PE}
        ;FOLD Parameters ;%{h}
        ;Params IlfProvider=kukaroboter.basistech.inlineforms.movement.spline; Kuka.IsGlobalPoint=False; Kuka.PointName=P106; Kuka.BlendingEnabled=False; Kuka.MoveDataName=CPDAT28; Kuka.VelocityPath=0.1; Kuka.VelocityFieldEnabled=True; Kuka.ColDetectFieldEnabled=True; Kuka.CurrentCDSetIndex=0; Kuka.MovementParameterFieldEnabled=True; IlfCommand=SLIN
        ;ENDFOLD
        SLIN XP106 WITH $VEL = SVEL_CP(0.1, , LCPDAT28), $TOOL = STOOL2(FP106), $BASE = SBASE(FP106.BASE_NO), $IPO_MODE = SIPO_MODE(FP106.IPO_FRAME), $LOAD = SLOAD(FP106.TOOL_NO), $ACC = SACC_CP(LCPDAT28), $ORI_TYPE = SORI_TYP(LCPDAT28), $APO = SAPO(LCPDAT28), $JERK = SJERK(LCPDAT28), $COLLMON_TOL_PRO[1] = USE_CM_PRO_VALUES(0)
        ;ENDFOLD
      ENDIF

      IF initialPosition == 7 THEN
        ;FOLD SPTP P107 Vel=100 % PDAT1 Tool[1]:SMC Base[0] ;%{PE}
        ;FOLD Parameters ;%{h}
        ;Params IlfProvider=kukaroboter.basistech.inlineforms.movement.spline; Kuka.IsGlobalPoint=False; Kuka.PointName=P107; Kuka.BlendingEnabled=False; Kuka.MoveDataPtpName=PDAT1; Kuka.VelocityPtp=100; Kuka.VelocityFieldEnabled=True; Kuka.ColDetectFieldEnabled=True; Kuka.CurrentCDSetIndex=0; Kuka.MovementParameterFieldEnabled=True; IlfCommand=SPTP
        ;ENDFOLD
        SPTP XP107 WITH $VEL_AXIS[1] = SVEL_JOINT(100.0), $TOOL = STOOL2(FP107), $BASE = SBASE(FP107.BASE_NO), $IPO_MODE = SIPO_MODE(FP107.IPO_FRAME), $LOAD = SLOAD(FP107.TOOL_NO), $ACC_AXIS[1] = SACC_JOINT(PPDAT1), $APO = SAPO_PTP(PPDAT1), $GEAR_JERK[1] = SGEAR_JERK(PPDAT1), $COLLMON_TOL_PRO[1] = USE_CM_PRO_VALUES(0)
        ;ENDFOLD
        ;FOLD SLIN P207 Vel=0.1 m/s CPDAT27 Tool[1]:SMC Base[0] ;%{PE}
        ;FOLD Parameters ;%{h}
        ;Params IlfProvider=kukaroboter.basistech.inlineforms.movement.spline; Kuka.IsGlobalPoint=False; Kuka.PointName=P207; Kuka.BlendingEnabled=False; Kuka.MoveDataName=CPDAT27; Kuka.VelocityPath=0.1; Kuka.VelocityFieldEnabled=True; Kuka.ColDetectFieldEnabled=True; Kuka.CurrentCDSetIndex=0; Kuka.MovementParameterFieldEnabled=True; IlfCommand=SLIN
        ;ENDFOLD
        SLIN XP207 WITH $VEL = SVEL_CP(0.1, , LCPDAT27), $TOOL = STOOL2(FP207), $BASE = SBASE(FP207.BASE_NO), $IPO_MODE = SIPO_MODE(FP207.IPO_FRAME), $LOAD = SLOAD(FP207.TOOL_NO), $ACC = SACC_CP(LCPDAT27), $ORI_TYPE = SORI_TYP(LCPDAT27), $APO = SAPO(LCPDAT27), $JERK = SJERK(LCPDAT27), $COLLMON_TOL_PRO[1] = USE_CM_PRO_VALUES(0)
        ;ENDFOLD
        ;FOLD Gripper SET [1]Gripper1 State=[2]CERRADA Wait 0.2[s] Check with Strategy 1 ;%{PE}
        ;FOLD Parameters Parameters ;%{h}
        ;Params IlfProvider=GripperTech.GripperSet;setgripper=1;setstate=2;setcont=nocont;waittime=0.2;errorstrategy=1
        ;ENDFOLD
        GRPg_SetStateAndCheck(1, 2, 0.2, 1)
        ;ENDFOLD
        ;FOLD SLIN P107 Vel=0.1 m/s CPDAT28 Tool[1]:SMC Base[0] ;%{PE}
        ;FOLD Parameters ;%{h}
        ;Params IlfProvider=kukaroboter.basistech.inlineforms.movement.spline; Kuka.IsGlobalPoint=False; Kuka.PointName=P107; Kuka.BlendingEnabled=False; Kuka.MoveDataName=CPDAT28; Kuka.VelocityPath=0.1; Kuka.VelocityFieldEnabled=True; Kuka.ColDetectFieldEnabled=True; Kuka.CurrentCDSetIndex=0; Kuka.MovementParameterFieldEnabled=True; IlfCommand=SLIN
        ;ENDFOLD
        SLIN XP107 WITH $VEL = SVEL_CP(0.1, , LCPDAT28), $TOOL = STOOL2(FP107), $BASE = SBASE(FP107.BASE_NO), $IPO_MODE = SIPO_MODE(FP107.IPO_FRAME), $LOAD = SLOAD(FP107.TOOL_NO), $ACC = SACC_CP(LCPDAT28), $ORI_TYPE = SORI_TYP(LCPDAT28), $APO = SAPO(LCPDAT28), $JERK = SJERK(LCPDAT28), $COLLMON_TOL_PRO[1] = USE_CM_PRO_VALUES(0)
        ;ENDFOLD
      ENDIF

      IF initialPosition == 8 THEN
        ;FOLD SPTP P108 Vel=100 % PDAT1 Tool[1]:SMC Base[0] ;%{PE}
        ;FOLD Parameters ;%{h}
        ;Params IlfProvider=kukaroboter.basistech.inlineforms.movement.spline; Kuka.IsGlobalPoint=False; Kuka.PointName=P108; Kuka.BlendingEnabled=False; Kuka.MoveDataPtpName=PDAT1; Kuka.VelocityPtp=100; Kuka.VelocityFieldEnabled=True; Kuka.ColDetectFieldEnabled=True; Kuka.CurrentCDSetIndex=0; Kuka.MovementParameterFieldEnabled=True; IlfCommand=SPTP
        ;ENDFOLD
        SPTP XP108 WITH $VEL_AXIS[1] = SVEL_JOINT(100.0), $TOOL = STOOL2(FP108), $BASE = SBASE(FP108.BASE_NO), $IPO_MODE = SIPO_MODE(FP108.IPO_FRAME), $LOAD = SLOAD(FP108.TOOL_NO), $ACC_AXIS[1] = SACC_JOINT(PPDAT1), $APO = SAPO_PTP(PPDAT1), $GEAR_JERK[1] = SGEAR_JERK(PPDAT1), $COLLMON_TOL_PRO[1] = USE_CM_PRO_VALUES(0)
        ;ENDFOLD
        ;FOLD SLIN P208 Vel=0.1 m/s CPDAT27 Tool[1]:SMC Base[0] ;%{PE}
        ;FOLD Parameters ;%{h}
        ;Params IlfProvider=kukaroboter.basistech.inlineforms.movement.spline; Kuka.IsGlobalPoint=False; Kuka.PointName=P208; Kuka.BlendingEnabled=False; Kuka.MoveDataName=CPDAT27; Kuka.VelocityPath=0.1; Kuka.VelocityFieldEnabled=True; Kuka.ColDetectFieldEnabled=True; Kuka.CurrentCDSetIndex=0; Kuka.MovementParameterFieldEnabled=True; IlfCommand=SLIN
        ;ENDFOLD
        SLIN XP208 WITH $VEL = SVEL_CP(0.1, , LCPDAT27), $TOOL = STOOL2(FP208), $BASE = SBASE(FP208.BASE_NO), $IPO_MODE = SIPO_MODE(FP208.IPO_FRAME), $LOAD = SLOAD(FP208.TOOL_NO), $ACC = SACC_CP(LCPDAT27), $ORI_TYPE = SORI_TYP(LCPDAT27), $APO = SAPO(LCPDAT27), $JERK = SJERK(LCPDAT27), $COLLMON_TOL_PRO[1] = USE_CM_PRO_VALUES(0)
        ;ENDFOLD
        ;FOLD Gripper SET [1]Gripper1 State=[2]CERRADA Wait 0.2[s] Check with Strategy 1 ;%{PE}
        ;FOLD Parameters Parameters ;%{h}
        ;Params IlfProvider=GripperTech.GripperSet;setgripper=1;setstate=2;setcont=nocont;waittime=0.2;errorstrategy=1
        ;ENDFOLD
        GRPg_SetStateAndCheck(1, 2, 0.2, 1)
        ;ENDFOLD
        ;FOLD SLIN P108 Vel=0.1 m/s CPDAT28 Tool[1]:SMC Base[0] ;%{PE}
        ;FOLD Parameters ;%{h}
        ;Params IlfProvider=kukaroboter.basistech.inlineforms.movement.spline; Kuka.IsGlobalPoint=False; Kuka.PointName=P108; Kuka.BlendingEnabled=False; Kuka.MoveDataName=CPDAT28; Kuka.VelocityPath=0.1; Kuka.VelocityFieldEnabled=True; Kuka.ColDetectFieldEnabled=True; Kuka.CurrentCDSetIndex=0; Kuka.MovementParameterFieldEnabled=True; IlfCommand=SLIN
        ;ENDFOLD
        SLIN XP108 WITH $VEL = SVEL_CP(0.1, , LCPDAT28), $TOOL = STOOL2(FP108), $BASE = SBASE(FP108.BASE_NO), $IPO_MODE = SIPO_MODE(FP108.IPO_FRAME), $LOAD = SLOAD(FP108.TOOL_NO), $ACC = SACC_CP(LCPDAT28), $ORI_TYPE = SORI_TYP(LCPDAT28), $APO = SAPO(LCPDAT28), $JERK = SJERK(LCPDAT28), $COLLMON_TOL_PRO[1] = USE_CM_PRO_VALUES(0)
        ;ENDFOLD
      ENDIF

      IF initialPosition == 9 THEN
        ;FOLD SPTP P109 Vel=100 % PDAT1 Tool[1]:SMC Base[0] ;%{PE}
        ;FOLD Parameters ;%{h}
        ;Params IlfProvider=kukaroboter.basistech.inlineforms.movement.spline; Kuka.IsGlobalPoint=False; Kuka.PointName=P109; Kuka.BlendingEnabled=False; Kuka.MoveDataPtpName=PDAT1; Kuka.VelocityPtp=100; Kuka.VelocityFieldEnabled=True; Kuka.ColDetectFieldEnabled=True; Kuka.CurrentCDSetIndex=0; Kuka.MovementParameterFieldEnabled=True; IlfCommand=SPTP
        ;ENDFOLD
        SPTP XP109 WITH $VEL_AXIS[1] = SVEL_JOINT(100.0), $TOOL = STOOL2(FP109), $BASE = SBASE(FP109.BASE_NO), $IPO_MODE = SIPO_MODE(FP109.IPO_FRAME), $LOAD = SLOAD(FP109.TOOL_NO), $ACC_AXIS[1] = SACC_JOINT(PPDAT1), $APO = SAPO_PTP(PPDAT1), $GEAR_JERK[1] = SGEAR_JERK(PPDAT1), $COLLMON_TOL_PRO[1] = USE_CM_PRO_VALUES(0)
        ;ENDFOLD
        ;FOLD SLIN P209 Vel=0.1 m/s CPDAT27 Tool[1]:SMC Base[0] ;%{PE}
        ;FOLD Parameters ;%{h}
        ;Params IlfProvider=kukaroboter.basistech.inlineforms.movement.spline; Kuka.IsGlobalPoint=False; Kuka.PointName=P209; Kuka.BlendingEnabled=False; Kuka.MoveDataName=CPDAT27; Kuka.VelocityPath=0.1; Kuka.VelocityFieldEnabled=True; Kuka.ColDetectFieldEnabled=True; Kuka.CurrentCDSetIndex=0; Kuka.MovementParameterFieldEnabled=True; IlfCommand=SLIN
        ;ENDFOLD
        SLIN XP209 WITH $VEL = SVEL_CP(0.1, , LCPDAT27), $TOOL = STOOL2(FP209), $BASE = SBASE(FP209.BASE_NO), $IPO_MODE = SIPO_MODE(FP209.IPO_FRAME), $LOAD = SLOAD(FP209.TOOL_NO), $ACC = SACC_CP(LCPDAT27), $ORI_TYPE = SORI_TYP(LCPDAT27), $APO = SAPO(LCPDAT27), $JERK = SJERK(LCPDAT27), $COLLMON_TOL_PRO[1] = USE_CM_PRO_VALUES(0)
        ;ENDFOLD
        ;FOLD Gripper SET [1]Gripper1 State=[2]CERRADA Wait 0.2[s] Check with Strategy 1 ;%{PE}
        ;FOLD Parameters Parameters ;%{h}
        ;Params IlfProvider=GripperTech.GripperSet;setgripper=1;setstate=2;setcont=nocont;waittime=0.2;errorstrategy=1
        ;ENDFOLD
        GRPg_SetStateAndCheck(1, 2, 0.2, 1)
        ;ENDFOLD
        ;FOLD SLIN P109 Vel=0.1 m/s CPDAT28 Tool[1]:SMC Base[0] ;%{PE}
        ;FOLD Parameters ;%{h}
        ;Params IlfProvider=kukaroboter.basistech.inlineforms.movement.spline; Kuka.IsGlobalPoint=False; Kuka.PointName=P109; Kuka.BlendingEnabled=False; Kuka.MoveDataName=CPDAT28; Kuka.VelocityPath=0.1; Kuka.VelocityFieldEnabled=True; Kuka.ColDetectFieldEnabled=True; Kuka.CurrentCDSetIndex=0; Kuka.MovementParameterFieldEnabled=True; IlfCommand=SLIN
        ;ENDFOLD
        SLIN XP109 WITH $VEL = SVEL_CP(0.1, , LCPDAT28), $TOOL = STOOL2(FP109), $BASE = SBASE(FP109.BASE_NO), $IPO_MODE = SIPO_MODE(FP109.IPO_FRAME), $LOAD = SLOAD(FP109.TOOL_NO), $ACC = SACC_CP(LCPDAT28), $ORI_TYPE = SORI_TYP(LCPDAT28), $APO = SAPO(LCPDAT28), $JERK = SJERK(LCPDAT28), $COLLMON_TOL_PRO[1] = USE_CM_PRO_VALUES(0)
        ;ENDFOLD
      ENDIF

      IF initialPosition == 10 THEN
        ;FOLD SPTP P110 Vel=100 % PDAT1 Tool[1]:SMC Base[0] ;%{PE}
        ;FOLD Parameters ;%{h}
        ;Params IlfProvider=kukaroboter.basistech.inlineforms.movement.spline; Kuka.IsGlobalPoint=False; Kuka.PointName=P110; Kuka.BlendingEnabled=False; Kuka.MoveDataPtpName=PDAT1; Kuka.VelocityPtp=100; Kuka.VelocityFieldEnabled=True; Kuka.ColDetectFieldEnabled=True; Kuka.CurrentCDSetIndex=0; Kuka.MovementParameterFieldEnabled=True; IlfCommand=SPTP
        ;ENDFOLD
        SPTP XP110 WITH $VEL_AXIS[1] = SVEL_JOINT(100.0), $TOOL = STOOL2(FP110), $BASE = SBASE(FP110.BASE_NO), $IPO_MODE = SIPO_MODE(FP110.IPO_FRAME), $LOAD = SLOAD(FP110.TOOL_NO), $ACC_AXIS[1] = SACC_JOINT(PPDAT1), $APO = SAPO_PTP(PPDAT1), $GEAR_JERK[1] = SGEAR_JERK(PPDAT1), $COLLMON_TOL_PRO[1] = USE_CM_PRO_VALUES(0)
        ;ENDFOLD
        ;FOLD SLIN P210 Vel=0.1 m/s CPDAT27 Tool[1]:SMC Base[0] ;%{PE}
        ;FOLD Parameters ;%{h}
        ;Params IlfProvider=kukaroboter.basistech.inlineforms.movement.spline; Kuka.IsGlobalPoint=False; Kuka.PointName=P210; Kuka.BlendingEnabled=False; Kuka.MoveDataName=CPDAT27; Kuka.VelocityPath=0.1; Kuka.VelocityFieldEnabled=True; Kuka.ColDetectFieldEnabled=True; Kuka.CurrentCDSetIndex=0; Kuka.MovementParameterFieldEnabled=True; IlfCommand=SLIN
        ;ENDFOLD
        SLIN XP210 WITH $VEL = SVEL_CP(0.1, , LCPDAT27), $TOOL = STOOL2(FP210), $BASE = SBASE(FP210.BASE_NO), $IPO_MODE = SIPO_MODE(FP210.IPO_FRAME), $LOAD = SLOAD(FP210.TOOL_NO), $ACC = SACC_CP(LCPDAT27), $ORI_TYPE = SORI_TYP(LCPDAT27), $APO = SAPO(LCPDAT27), $JERK = SJERK(LCPDAT27), $COLLMON_TOL_PRO[1] = USE_CM_PRO_VALUES(0)
        ;ENDFOLD
        ;FOLD Gripper SET [1]Gripper1 State=[2]CERRADA Wait 0.2[s] Check with Strategy 1 ;%{PE}
        ;FOLD Parameters Parameters ;%{h}
        ;Params IlfProvider=GripperTech.GripperSet;setgripper=1;setstate=2;setcont=nocont;waittime=0.2;errorstrategy=1
        ;ENDFOLD
        GRPg_SetStateAndCheck(1, 2, 0.2, 1)
        ;ENDFOLD
        ;FOLD SLIN P110 Vel=0.1 m/s CPDAT28 Tool[1]:SMC Base[0] ;%{PE}
        ;FOLD Parameters ;%{h}
        ;Params IlfProvider=kukaroboter.basistech.inlineforms.movement.spline; Kuka.IsGlobalPoint=False; Kuka.PointName=P110; Kuka.BlendingEnabled=False; Kuka.MoveDataName=CPDAT28; Kuka.VelocityPath=0.1; Kuka.VelocityFieldEnabled=True; Kuka.ColDetectFieldEnabled=True; Kuka.CurrentCDSetIndex=0; Kuka.MovementParameterFieldEnabled=True; IlfCommand=SLIN
        ;ENDFOLD
        SLIN XP110 WITH $VEL = SVEL_CP(0.1, , LCPDAT28), $TOOL = STOOL2(FP110), $BASE = SBASE(FP110.BASE_NO), $IPO_MODE = SIPO_MODE(FP110.IPO_FRAME), $LOAD = SLOAD(FP110.TOOL_NO), $ACC = SACC_CP(LCPDAT28), $ORI_TYPE = SORI_TYP(LCPDAT28), $APO = SAPO(LCPDAT28), $JERK = SJERK(LCPDAT28), $COLLMON_TOL_PRO[1] = USE_CM_PRO_VALUES(0)
        ;ENDFOLD
      ENDIF

      IF initialPosition == 11 THEN
        ;FOLD SPTP P111 Vel=100 % PDAT1 Tool[1]:SMC Base[0] ;%{PE}
        ;FOLD Parameters ;%{h}
        ;Params IlfProvider=kukaroboter.basistech.inlineforms.movement.spline; Kuka.IsGlobalPoint=False; Kuka.PointName=P111; Kuka.BlendingEnabled=False; Kuka.MoveDataPtpName=PDAT1; Kuka.VelocityPtp=100; Kuka.VelocityFieldEnabled=True; Kuka.ColDetectFieldEnabled=True; Kuka.CurrentCDSetIndex=0; Kuka.MovementParameterFieldEnabled=True; IlfCommand=SPTP
        ;ENDFOLD
        SPTP XP111 WITH $VEL_AXIS[1] = SVEL_JOINT(100.0), $TOOL = STOOL2(FP111), $BASE = SBASE(FP111.BASE_NO), $IPO_MODE = SIPO_MODE(FP111.IPO_FRAME), $LOAD = SLOAD(FP111.TOOL_NO), $ACC_AXIS[1] = SACC_JOINT(PPDAT1), $APO = SAPO_PTP(PPDAT1), $GEAR_JERK[1] = SGEAR_JERK(PPDAT1), $COLLMON_TOL_PRO[1] = USE_CM_PRO_VALUES(0)
        ;ENDFOLD
        ;FOLD SLIN P211 Vel=0.1 m/s CPDAT27 Tool[1]:SMC Base[0] ;%{PE}
        ;FOLD Parameters ;%{h}
        ;Params IlfProvider=kukaroboter.basistech.inlineforms.movement.spline; Kuka.IsGlobalPoint=False; Kuka.PointName=P211; Kuka.BlendingEnabled=False; Kuka.MoveDataName=CPDAT27; Kuka.VelocityPath=0.1; Kuka.VelocityFieldEnabled=True; Kuka.ColDetectFieldEnabled=True; Kuka.CurrentCDSetIndex=0; Kuka.MovementParameterFieldEnabled=True; IlfCommand=SLIN
        ;ENDFOLD
        SLIN XP211 WITH $VEL = SVEL_CP(0.1, , LCPDAT27), $TOOL = STOOL2(FP211), $BASE = SBASE(FP211.BASE_NO), $IPO_MODE = SIPO_MODE(FP211.IPO_FRAME), $LOAD = SLOAD(FP211.TOOL_NO), $ACC = SACC_CP(LCPDAT27), $ORI_TYPE = SORI_TYP(LCPDAT27), $APO = SAPO(LCPDAT27), $JERK = SJERK(LCPDAT27), $COLLMON_TOL_PRO[1] = USE_CM_PRO_VALUES(0)
        ;ENDFOLD
        ;FOLD Gripper SET [1]Gripper1 State=[2]CERRADA Wait 0.2[s] Check with Strategy 1 ;%{PE}
        ;FOLD Parameters Parameters ;%{h}
        ;Params IlfProvider=GripperTech.GripperSet;setgripper=1;setstate=2;setcont=nocont;waittime=0.2;errorstrategy=1
        ;ENDFOLD
        GRPg_SetStateAndCheck(1, 2, 0.2, 1)
        ;ENDFOLD
        ;FOLD SLIN P111 Vel=0.1 m/s CPDAT28 Tool[1]:SMC Base[0] ;%{PE}
        ;FOLD Parameters ;%{h}
        ;Params IlfProvider=kukaroboter.basistech.inlineforms.movement.spline; Kuka.IsGlobalPoint=False; Kuka.PointName=P111; Kuka.BlendingEnabled=False; Kuka.MoveDataName=CPDAT28; Kuka.VelocityPath=0.1; Kuka.VelocityFieldEnabled=True; Kuka.ColDetectFieldEnabled=True; Kuka.CurrentCDSetIndex=0; Kuka.MovementParameterFieldEnabled=True; IlfCommand=SLIN
        ;ENDFOLD
        SLIN XP111 WITH $VEL = SVEL_CP(0.1, , LCPDAT28), $TOOL = STOOL2(FP111), $BASE = SBASE(FP111.BASE_NO), $IPO_MODE = SIPO_MODE(FP111.IPO_FRAME), $LOAD = SLOAD(FP111.TOOL_NO), $ACC = SACC_CP(LCPDAT28), $ORI_TYPE = SORI_TYP(LCPDAT28), $APO = SAPO(LCPDAT28), $JERK = SJERK(LCPDAT28), $COLLMON_TOL_PRO[1] = USE_CM_PRO_VALUES(0)
        ;ENDFOLD
      ENDIF

      IF initialPosition == 12 THEN
        ;FOLD SPTP P112 Vel=100 % PDAT1 Tool[1]:SMC Base[0] ;%{PE}
        ;FOLD Parameters ;%{h}
        ;Params IlfProvider=kukaroboter.basistech.inlineforms.movement.spline; Kuka.IsGlobalPoint=False; Kuka.PointName=P112; Kuka.BlendingEnabled=False; Kuka.MoveDataPtpName=PDAT1; Kuka.VelocityPtp=100; Kuka.VelocityFieldEnabled=True; Kuka.ColDetectFieldEnabled=True; Kuka.CurrentCDSetIndex=0; Kuka.MovementParameterFieldEnabled=True; IlfCommand=SPTP
        ;ENDFOLD
        SPTP XP112 WITH $VEL_AXIS[1] = SVEL_JOINT(100.0), $TOOL = STOOL2(FP112), $BASE = SBASE(FP112.BASE_NO), $IPO_MODE = SIPO_MODE(FP112.IPO_FRAME), $LOAD = SLOAD(FP112.TOOL_NO), $ACC_AXIS[1] = SACC_JOINT(PPDAT1), $APO = SAPO_PTP(PPDAT1), $GEAR_JERK[1] = SGEAR_JERK(PPDAT1), $COLLMON_TOL_PRO[1] = USE_CM_PRO_VALUES(0)
        ;ENDFOLD
        ;FOLD SLIN P212 Vel=0.1 m/s CPDAT27 Tool[1]:SMC Base[0] ;%{PE}
        ;FOLD Parameters ;%{h}
        ;Params IlfProvider=kukaroboter.basistech.inlineforms.movement.spline; Kuka.IsGlobalPoint=False; Kuka.PointName=P212; Kuka.BlendingEnabled=False; Kuka.MoveDataName=CPDAT27; Kuka.VelocityPath=0.1; Kuka.VelocityFieldEnabled=True; Kuka.ColDetectFieldEnabled=True; Kuka.CurrentCDSetIndex=0; Kuka.MovementParameterFieldEnabled=True; IlfCommand=SLIN
        ;ENDFOLD
        SLIN XP212 WITH $VEL = SVEL_CP(0.1, , LCPDAT27), $TOOL = STOOL2(FP212), $BASE = SBASE(FP212.BASE_NO), $IPO_MODE = SIPO_MODE(FP212.IPO_FRAME), $LOAD = SLOAD(FP212.TOOL_NO), $ACC = SACC_CP(LCPDAT27), $ORI_TYPE = SORI_TYP(LCPDAT27), $APO = SAPO(LCPDAT27), $JERK = SJERK(LCPDAT27), $COLLMON_TOL_PRO[1] = USE_CM_PRO_VALUES(0)
        ;ENDFOLD
        ;FOLD Gripper SET [1]Gripper1 State=[2]CERRADA Wait 0.2[s] Check with Strategy 1 ;%{PE}
        ;FOLD Parameters Parameters ;%{h}
        ;Params IlfProvider=GripperTech.GripperSet;setgripper=1;setstate=2;setcont=nocont;waittime=0.2;errorstrategy=1
        ;ENDFOLD
        GRPg_SetStateAndCheck(1, 2, 0.2, 1)
        ;ENDFOLD
        ;FOLD SLIN P112 Vel=0.1 m/s CPDAT28 Tool[1]:SMC Base[0] ;%{PE}
        ;FOLD Parameters ;%{h}
        ;Params IlfProvider=kukaroboter.basistech.inlineforms.movement.spline; Kuka.IsGlobalPoint=False; Kuka.PointName=P112; Kuka.BlendingEnabled=False; Kuka.MoveDataName=CPDAT28; Kuka.VelocityPath=0.1; Kuka.VelocityFieldEnabled=True; Kuka.ColDetectFieldEnabled=True; Kuka.CurrentCDSetIndex=0; Kuka.MovementParameterFieldEnabled=True; IlfCommand=SLIN
        ;ENDFOLD
        SLIN XP112 WITH $VEL = SVEL_CP(0.1, , LCPDAT28), $TOOL = STOOL2(FP112), $BASE = SBASE(FP112.BASE_NO), $IPO_MODE = SIPO_MODE(FP112.IPO_FRAME), $LOAD = SLOAD(FP112.TOOL_NO), $ACC = SACC_CP(LCPDAT28), $ORI_TYPE = SORI_TYP(LCPDAT28), $APO = SAPO(LCPDAT28), $JERK = SJERK(LCPDAT28), $COLLMON_TOL_PRO[1] = USE_CM_PRO_VALUES(0)
        ;ENDFOLD
      ENDIF

